gfCNCPoint3[4861] = {X 137.2439, Y 19.5606, Z -3.8333, A 0.000, B 0.000, C 0.000 }
gfCNCPoint3[4862] = {X 137.1370, Y 19.7298, Z -3.8333, A 0.000, B 0.000, C 0.000 }
gfCNCPoint3[4863] = {X 136.4975, Y 20.4532, Z -3.8333, A 0.000, B 0.000, C 0.000 }
gfCNCPoint3[4864] = {X 135.7033, Y 21.0023, Z -3.8333, A 0.000, B 0.000, C 0.000 }
gfCNCPoint3[4865] = {X 134.8007, Y 21.3450, Z -3.8333, A 0.000, B 0.000, C 0.000 }
gfCNCPoint3[4866] = {X 133.8422, Y 21.4615, Z -3.8333, A 0.000, B 0.000, C 0.000 }
gfCNCPoint3[4867] = {X 133.2006, Y 21.4615, Z -3.8333, A 0.000, B 0.000, C 0.000 }
gfCNCPoint3[4868] = {X 132.3106, Y 21.3612, Z -3.8333, A 0.000, B 0.000, C 0.000 }
gfCNCPoint3[4869] = {X 131.4651, Y 21.0654, Z -3.8333, A 0.000, B 0.000, C 0.000 }
gfCNCPoint3[4870] = {X 130.7067, Y 20.5889, Z -3.8333, A 0.000, B 0.000, C 0.000 }
gfCNCPoint3[4871] = {X 130.0733, Y 19.9555, Z -3.8333, A 0.000, B 0.000, C 0.000 }
gfCNCPoint3[4872] = {X 129.5968, Y 19.1971, Z -3.8333, A 0.000, B 0.000, C 0.000 }
gfCNCPoint3[4873] = {X 129.3009, Y 18.3516, Z -3.8333, A 0.000, B 0.000, C 0.000 }
gfCNCPoint3[4874] = {X 129.2006, Y 17.4615, Z -3.8333, A 0.000, B 0.000, C 0.000 }
gfCNCPoint3[4875] = {X 129.2006, Y 10.4835, Z -3.8333, A 0.000, B 0.000, C 0.000 }
gfCNCPoint3[4876] = {X 129.3009, Y 9.5934, Z -3.8333, A 0.000, B 0.000, C 0.000 }
gfCNCPoint3[4877] = {X 129.5968, Y 8.7480, Z -3.8333, A 0.000, B 0.000, C 0.000 }
gfCNCPoint3[4878] = {X 130.0733, Y 7.9895, Z -3.8333, A 0.000, B 0.000, C 0.000 }
gfCNCPoint3[4879] = {X 130.7067, Y 7.3562, Z -3.8333, A 0.000, B 0.000, C 0.000 }
gfCNCPoint3[4880] = {X 131.4651, Y 6.8796, Z -3.8333, A 0.000, B 0.000, C 0.000 }
gfCNCPoint3[4881] = {X 132.3106, Y 6.5838, Z -3.8333, A 0.000, B 0.000, C 0.000 }
gfCNCPoint3[4882] = {X 133.2007, Y 6.4835, Z -3.8333, A 0.000, B 0.000, C 0.000 }
gfCNCPoint3[4883] = {X 133.8833, Y 6.4837, Z -3.8333, A 0.000, B 0.000, C 0.000 }
gfCNCPoint3[4884] = {X 134.6794, Y 6.5721, Z -3.8333, A 0.000, B 0.000, C 0.000 }
gfCNCPoint3[4885] = {X 135.4419, Y 6.8173, Z -3.8333, A 0.000, B 0.000, C 0.000 }
gfCNCPoint3[4886] = {X 136.1403, Y 7.2095, Z -3.8333, A 0.000, B 0.000, C 0.000 }
gfCNCPoint3[4887] = {X 136.7465, Y 7.7329, Z -3.8333, A 0.000, B 0.000, C 0.000 }
gfCNCPoint3[4888] = {X 137.2363, Y 8.3667, Z -3.8333, A 0.000, B 0.000, C 0.000 }
gfCNCPoint3[4889] = {X 155.2276, Y 8.3667, Z -3.8333, A 0.000, B 0.000, C 0.000 }
gfCNCPoint3[4890] = {X 155.2814, Y 8.3748, Z -3.8333, A 0.000, B 0.000, C 0.000 }
gfCNCPoint3[4891] = {X 155.3392, Y 8.2843, Z -3.8333, A 0.000, B 0.000, C 0.000 }
gfCNCPoint3[4892] = {X 155.3994, Y 8.1955, Z -3.8333, A 0.000, B 0.000, C 0.000 }
gfCNCPoint3[4893] = {X 156.0387, Y 7.4799, Z -3.8333, A 0.000, B 0.000, C 0.000 }
gfCNCPoint3[4894] = {X 156.8301, Y 6.9372, Z -3.8333, A 0.000, B 0.000, C 0.000 }
gfCNCPoint3[4895] = {X 157.7279, Y 6.5986, Z -3.8333, A 0.000, B 0.000, C 0.000 }
gfCNCPoint3[4896] = {X 158.6806, Y 6.4835, Z -3.8333, A 0.000, B 0.000, C 0.000 }
gfCNCPoint3[4897] = {X 159.3739, Y 6.4839, Z -3.8333, A 0.000, B 0.000, C 0.000 }
gfCNCPoint3[4898] = {X 160.2554, Y 6.5939, Z -3.8333, A 0.000, B 0.000, C 0.000 }
gfCNCPoint3[4899] = {X 161.0909, Y 6.8959, Z -3.8333, A 0.000, B 0.000, C 0.000 }
gfCNCPoint3[4900] = {X 161.8391, Y 7.3747, Z -3.8333, A 0.000, B 0.000, C 0.000 }
gfCNCPoint3[4901] = {X 162.4632, Y 8.0070, Z -3.8333, A 0.000, B 0.000, C 0.000 }
gfCNCPoint3[4902] = {X 162.9324, Y 8.7613, Z -3.8333, A 0.000, B 0.000, C 0.000 }
gfCNCPoint3[4903] = {X 163.2234, Y 9.6007, Z -3.8333, A 0.000, B 0.000, C 0.000 }
gfCNCPoint3[4904] = {X 163.3221, Y 10.4835, Z -3.8333, A 0.000, B 0.000, C 0.000 }
gfCNCPoint3[4905] = {X 163.3221, Y 17.4615, Z -3.8333, A 0.000, B 0.000, C 0.000 }
gfCNCPoint3[4906] = {X 163.2218, Y 18.3516, Z -3.8333, A 0.000, B 0.000, C 0.000 }
gfCNCPoint3[4907] = {X 162.9260, Y 19.1971, Z -3.8333, A 0.000, B 0.000, C 0.000 }
gfCNCPoint3[4908] = {X 162.4494, Y 19.9555, Z -3.8333, A 0.000, B 0.000, C 0.000 }
gfCNCPoint3[4909] = {X 161.8160, Y 20.5889, Z -3.8333, A 0.000, B 0.000, C 0.000 }
gfCNCPoint3[4910] = {X 161.0576, Y 21.0654, Z -3.8333, A 0.000, B 0.000, C 0.000 }
gfCNCPoint3[4911] = {X 160.2121, Y 21.3613, Z -3.8333, A 0.000, B 0.000, C 0.000 }
gfCNCPoint3[4912] = {X 159.3221, Y 21.4615, Z -3.8333, A 0.000, B 0.000, C 0.000 }
gfCNCPoint3[4913] = {X 158.6805, Y 21.4615, Z -3.8333, A 0.000, B 0.000, C 0.000 }
gfCNCPoint3[4914] = {X 157.8711, Y 21.3759, Z -3.8333, A 0.000, B 0.000, C 0.000 }
gfCNCPoint3[4915] = {X 157.0952, Y 21.1295, Z -3.8333, A 0.000, B 0.000, C 0.000 }
gfCNCPoint3[4916] = {X 156.3846, Y 20.7325, Z -3.8333, A 0.000, B 0.000, C 0.000 }
gfCNCPoint3[4917] = {X 155.7681, Y 20.2010, Z -3.8333, A 0.000, B 0.000, C 0.000 }
gfCNCPoint3[4918] = {X 155.2709, Y 19.5565, Z -3.8333, A 0.000, B 0.000, C 0.000 }
gfCNCPoint3[4919] = {X 151.9562, Y 19.5580, Z -3.8333, A 0.000, B 0.000, C 0.000 }
gfCNCPoint3[4920] = {X 151.9548, Y 40.9999, Z -3.8333, A 0.000, B 0.000, C 0.000 }
gfCNCPoint3[4921] = {X 152.5009, Y 41.5878, Z -3.8333, A 0.000, B 0.000, C 0.000 }
gfCNCPoint3[4922] = {X 152.5884, Y 41.6922, Z -3.8333, A 0.000, B 0.000, C 0.000 }
gfCNCPoint3[4923] = {X 153.0743, Y 42.4563, Z -3.8333, A 0.000, B 0.000, C 0.000 }
gfCNCPoint3[4924] = {X 153.3776, Y 43.3095, Z -3.8333, A 0.000, B 0.000, C 0.000 }
gfCNCPoint3[4925] = {X 153.4831, Y 44.2089, Z -3.8333, A 0.000, B 0.000, C 0.000 }
gfCNCPoint3[4926] = {X 153.4829, Y 45.0384, Z -3.8333, A 0.000, B 0.000, C 0.000 }
gfCNCPoint3[4927] = {X 153.3753, Y 45.9222, Z -3.8333, A 0.000, B 0.000, C 0.000 }
gfCNCPoint3[4928] = {X 153.0750, Y 46.7602, Z -3.8333, A 0.000, B 0.000, C 0.000 }
gfCNCPoint3[4929] = {X 152.5967, Y 47.5111, Z -3.8333, A 0.000, B 0.000, C 0.000 }
gfCNCPoint3[4930] = {X 151.9642, Y 48.1376, Z -3.8333, A 0.000, B 0.000, C 0.000 }
gfCNCPoint3[4931] = {X 151.2087, Y 48.6086, Z -3.8333, A 0.000, B 0.000, C 0.000 }
gfCNCPoint3[4932] = {X 150.3678, Y 48.9009, Z -3.8333, A 0.000, B 0.000, C 0.000 }
gfCNCPoint3[4933] = {X 149.4831, Y 49.0000, Z -3.8333, A 0.000, B 0.000, C 0.000 }
gfCNCPoint3[4934] = {X 143.0396, Y 49.0000, Z -3.8333, A 0.000, B 0.000, C 0.000 }
gfCNCPoint3[4935] = {X 142.1495, Y 48.8997, Z -3.8333, A 0.000, B 0.000, C 0.000 }
gfCNCPoint3[4936] = {X 141.3041, Y 48.6039, Z -3.8333, A 0.000, B 0.000, C 0.000 }
gfCNCPoint3[4937] = {X 140.5457, Y 48.1273, Z -3.8333, A 0.000, B 0.000, C 0.000 }
gfCNCPoint3[4938] = {X 139.9123, Y 47.4939, Z -3.8333, A 0.000, B 0.000, C 0.000 }
gfCNCPoint3[4939] = {X 139.4357, Y 46.7355, Z -3.8333, A 0.000, B 0.000, C 0.000 }
gfCNCPoint3[4940] = {X 139.1399, Y 45.8900, Z -3.8333, A 0.000, B 0.000, C 0.000 }
gfCNCPoint3[4941] = {X 139.0396, Y 45.0000, Z -3.8333, A 0.000, B 0.000, C 0.000 }
gfCNCPoint3[4942] = {X 139.0400, Y 44.1538, Z -3.8333, A 0.000, B 0.000, C 0.000 }
gfCNCPoint3[4943] = {X 139.1506, Y 43.2730, Z -3.8333, A 0.000, B 0.000, C 0.000 }
gfCNCPoint3[4944] = {X 139.4528, Y 42.4382, Z -3.8333, A 0.000, B 0.000, C 0.000 }
gfCNCPoint3[4945] = {X 139.9317, Y 41.6907, Z -3.8333, A 0.000, B 0.000, C 0.000 }
gfCNCPoint3[4946] = {X 140.5636, Y 41.0672, Z -3.8333, A 0.000, B 0.000, C 0.000 }
gfCNCPoint3[4947] = {X 140.5636, Y 30.3965, Z -3.8333, A 0.000, B 0.000, C 0.000 }
gfCNCPoint3[4948] = {X 136.4836, Y 30.3965, Z -3.8333, A 0.000, B 0.000, C 0.000 }
gfCNCPoint3[4949] = {X 136.4836, Y 30.3965, Z -0.8333, A 0.000, B 0.000, C 0.000 }
gfCNCPoint3[4950] = {X 136.4836, Y 30.3965, Z 11.0000, A 0.000, B 0.000, C 0.000 }
gfCNCPoint3[4951] = {X 137.6636, Y 74.8930, Z 11.0000, A 0.000, B 0.000, C 0.000 }
gfCNCPoint3[4952] = {X 137.6636, Y 74.8930, Z -0.8333, A 0.000, B 0.000, C 0.000 }
gfCNCPoint3[4953] = {X 137.6636, Y 74.8930, Z -3.8333, A 0.000, B 0.000, C 0.000 }
gfCNCPoint3[4954] = {X 140.6803, Y 77.6400, Z -3.8333, A 0.000, B 0.000, C 0.000 }
gfCNCPoint3[4955] = {X 155.6326, Y 61.2204, Z -3.8333, A 0.000, B 0.000, C 0.000 }
gfCNCPoint3[4956] = {X 155.2775, Y 60.5146, Z -3.8333, A 0.000, B 0.000, C 0.000 }
gfCNCPoint3[4957] = {X 155.0569, Y 59.7559, Z -3.8333, A 0.000, B 0.000, C 0.000 }
gfCNCPoint3[4958] = {X 154.9781, Y 58.9697, Z -3.8333, A 0.000, B 0.000, C 0.000 }
gfCNCPoint3[4959] = {X 154.9780, Y 58.0000, Z -3.8333, A 0.000, B 0.000, C 0.000 }
gfCNCPoint3[4960] = {X 155.0863, Y 57.0387, Z -3.8333, A 0.000, B 0.000, C 0.000 }
gfCNCPoint3[4961] = {X 155.4058, Y 56.1256, Z -3.8333, A 0.000, B 0.000, C 0.000 }
gfCNCPoint3[4962] = {X 155.9204, Y 55.3065, Z -3.8333, A 0.000, B 0.000, C 0.000 }
gfCNCPoint3[4963] = {X 156.6045, Y 54.6225, Z -3.8333, A 0.000, B 0.000, C 0.000 }
gfCNCPoint3[4964] = {X 157.4236, Y 54.1078, Z -3.8333, A 0.000, B 0.000, C 0.000 }
gfCNCPoint3[4965] = {X 158.3367, Y 53.7883, Z -3.8333, A 0.000, B 0.000, C 0.000 }
gfCNCPoint3[4966] = {X 159.2980, Y 53.6800, Z -3.8333, A 0.000, B 0.000, C 0.000 }
gfCNCPoint3[4967] = {X 178.5335, Y 53.6800, Z -3.8333, A 0.000, B 0.000, C 0.000 }
gfCNCPoint3[4968] = {X 179.4948, Y 53.7883, Z -3.8333, A 0.000, B 0.000, C 0.000 }
gfCNCPoint3[4969] = {X 180.4079, Y 54.1078, Z -3.8333, A 0.000, B 0.000, C 0.000 }
gfCNCPoint3[4970] = {X 181.2270, Y 54.6225, Z -3.8333, A 0.000, B 0.000, C 0.000 }
gfCNCPoint3[4971] = {X 181.9110, Y 55.3065, Z -3.8333, A 0.000, B 0.000, C 0.000 }
gfCNCPoint3[4972] = {X 182.4257, Y 56.1256, Z -3.8333, A 0.000, B 0.000, C 0.000 }
gfCNCPoint3[4973] = {X 182.7452, Y 57.0387, Z -3.8333, A 0.000, B 0.000, C 0.000 }
gfCNCPoint3[4974] = {X 182.8535, Y 58.0000, Z -3.8333, A 0.000, B 0.000, C 0.000 }
gfCNCPoint3[4975] = {X 182.8535, Y 58.9342, Z -3.8333, A 0.000, B 0.000, C 0.000 }
gfCNCPoint3[4976] = {X 182.7808, Y 59.7234, Z -3.8333, A 0.000, B 0.000, C 0.000 }
gfCNCPoint3[4977] = {X 182.5651, Y 60.4860, Z -3.8333, A 0.000, B 0.000, C 0.000 }
gfCNCPoint3[4978] = {X 182.2138, Y 61.1963, Z -3.8333, A 0.000, B 0.000, C 0.000 }
gfCNCPoint3[4979] = {X 209.4784, Y 90.9541, Z -3.8333, A 0.000, B 0.000, C 0.000 }
gfCNCPoint3[4980] = {X 210.1358, Y 91.6211, Z -3.8333, A 0.000, B 0.000, C 0.000 }
gfCNCPoint3[4981] = {X 210.8401, Y 92.2385, Z -3.8333, A 0.000, B 0.000, C 0.000 }
gfCNCPoint3[4982] = {X 211.1140, Y 92.4118, Z -3.8333, A 0.000, B 0.000, C 0.000 }
gfCNCPoint3[4983] = {X 211.4211, Y 92.5156, Z -3.8333, A 0.000, B 0.000, C 0.000 }
gfCNCPoint3[4984] = {X 213.4039, Y 92.8249, Z -3.8333, A 0.000, B 0.000, C 0.000 }
gfCNCPoint3[4985] = {X 214.4546, Y 92.7361, Z -3.8333, A 0.000, B 0.000, C 0.000 }
gfCNCPoint3[4986] = {X 215.5072, Y 92.6759, Z -3.8333, A 0.000, B 0.000, C 0.000 }
gfCNCPoint3[4987] = {X 216.1773, Y 92.6027, Z -3.8333, A 0.000, B 0.000, C 0.000 }
gfCNCPoint3[4988] = {X 216.8225, Y 92.4076, Z -3.8333, A 0.000, B 0.000, C 0.000 }
gfCNCPoint3[4989] = {X 217.4210, Y 92.0974, Z -3.8333, A 0.000, B 0.000, C 0.000 }
gfCNCPoint3[4990] = {X 222.9613, Y 88.5219, Z -3.8333, A 0.000, B 0.000, C 0.000 }
gfCNCPoint3[4991] = {X 245.8284, Y 73.8995, Z -3.8333, A 0.000, B 0.000, C 0.000 }
gfCNCPoint3[4992] = {X 221.6305, Y 64.4034, Z -3.8333, A 0.000, B 0.000, C 0.000 }
gfCNCPoint3[4993] = {X 219.8632, Y 63.8117, Z -3.8333, A 0.000, B 0.000, C 0.000 }
gfCNCPoint3[4994] = {X 218.0397, Y 63.4261, Z -3.8333, A 0.000, B 0.000, C 0.000 }
gfCNCPoint3[4995] = {X 216.1842, Y 63.2516, Z -3.8333, A 0.000, B 0.000, C 0.000 }
gfCNCPoint3[4996] = {X 215.2523, Y 63.1173, Z -3.8333, A 0.000, B 0.000, C 0.000 }
gfCNCPoint3[4997] = {X 214.3717, Y 62.7843, Z -3.8333, A 0.000, B 0.000, C 0.000 }
gfCNCPoint3[4998] = {X 213.5841, Y 62.2684, Z -3.8333, A 0.000, B 0.000, C 0.000 }
gfCNCPoint3[4999] = {X 212.9270, Y 61.5942, Z -3.8333, A 0.000, B 0.000, C 0.000 }
gfCNCPoint3[5000] = {X 212.4315, Y 60.7936, Z -3.8333, A 0.000, B 0.000, C 0.000 }
gfCNCPoint3[5001] = {X 212.1213, Y 59.9047, Z -3.8333, A 0.000, B 0.000, C 0.000 }
gfCNCPoint3[5002] = {X 212.0110, Y 58.9697, Z -3.8333, A 0.000, B 0.000, C 0.000 }
gfCNCPoint3[5003] = {X 212.0108, Y 58.0000, Z -3.8333, A 0.000, B 0.000, C 0.000 }
gfCNCPoint3[5004] = {X 212.1191, Y 57.0387, Z -3.8333, A 0.000, B 0.000, C 0.000 }
gfCNCPoint3[5005] = {X 212.4386, Y 56.1256, Z -3.8333, A 0.000, B 0.000, C 0.000 }
gfCNCPoint3[5006] = {X 212.9533, Y 55.3065, Z -3.8333, A 0.000, B 0.000, C 0.000 }
gfCNCPoint3[5007] = {X 213.6373, Y 54.6225, Z -3.8333, A 0.000, B 0.000, C 0.000 }
gfCNCPoint3[5008] = {X 214.4564, Y 54.1078, Z -3.8333, A 0.000, B 0.000, C 0.000 }
gfCNCPoint3[5009] = {X 215.3695, Y 53.7883, Z -3.8333, A 0.000, B 0.000, C 0.000 }
gfCNCPoint3[5010] = {X 216.3308, Y 53.6800, Z -3.8333, A 0.000, B 0.000, C 0.000 }
gfCNCPoint3[5011] = {X 237.2617, Y 53.6800, Z -3.8333, A 0.000, B 0.000, C 0.000 }
gfCNCPoint3[5012] = {X 238.2230, Y 53.7883, Z -3.8333, A 0.000, B 0.000, C 0.000 }
gfCNCPoint3[5013] = {X 239.1361, Y 54.1078, Z -3.8333, A 0.000, B 0.000, C 0.000 }
gfCNCPoint3[5014] = {X 239.9552, Y 54.6225, Z -3.8333, A 0.000, B 0.000, C 0.000 }
gfCNCPoint3[5015] = {X 240.6392, Y 55.3065, Z -3.8333, A 0.000, B 0.000, C 0.000 }
gfCNCPoint3[5016] = {X 241.1539, Y 56.1256, Z -3.8333, A 0.000, B 0.000, C 0.000 }
gfCNCPoint3[5017] = {X 241.4734, Y 57.0387, Z -3.8333, A 0.000, B 0.000, C 0.000 }
gfCNCPoint3[5018] = {X 241.5817, Y 58.0000, Z -3.8333, A 0.000, B 0.000, C 0.000 }
gfCNCPoint3[5019] = {X 241.5817, Y 58.2325, Z -3.8333, A 0.000, B 0.000, C 0.000 }
gfCNCPoint3[5020] = {X 247.4883, Y 60.5350, Z -3.8333, A 0.000, B 0.000, C 0.000 }
gfCNCPoint3[5021] = {X 275.6332, Y 71.7024, Z -3.8333, A 0.000, B 0.000, C 0.000 }
gfCNCPoint3[5022] = {X 275.6341, Y 63.2124, Z -3.8333, A 0.000, B 0.000, C 0.000 }
gfCNCPoint3[5023] = {X 274.7824, Y 63.0033, Z -3.8333, A 0.000, B 0.000, C 0.000 }
gfCNCPoint3[5024] = {X 273.9904, Y 62.6266, Z -3.8333, A 0.000, B 0.000, C 0.000 }
gfCNCPoint3[5025] = {X 273.2909, Y 62.0976, Z -3.8333, A 0.000, B 0.000, C 0.000 }
gfCNCPoint3[5026] = {X 272.7126, Y 61.4383, Z -3.8333, A 0.000, B 0.000, C 0.000 }
gfCNCPoint3[5027] = {X 272.2794, Y 60.6758, Z -3.8333, A 0.000, B 0.000, C 0.000 }
gfCNCPoint3[5028] = {X 272.0091, Y 59.8415, Z -3.8333, A 0.000, B 0.000, C 0.000 }
gfCNCPoint3[5029] = {X 271.9128, Y 58.9697, Z -3.8333, A 0.000, B 0.000, C 0.000 }
gfCNCPoint3[5030] = {X 271.9127, Y 58.0000, Z -3.8333, A 0.000, B 0.000, C 0.000 }
gfCNCPoint3[5031] = {X 272.0210, Y 57.0387, Z -3.8333, A 0.000, B 0.000, C 0.000 }
gfCNCPoint3[5032] = {X 272.3405, Y 56.1256, Z -3.8333, A 0.000, B 0.000, C 0.000 }
gfCNCPoint3[5033] = {X 272.8552, Y 55.3065, Z -3.8333, A 0.000, B 0.000, C 0.000 }
gfCNCPoint3[5034] = {X 273.5392, Y 54.6225, Z -3.8333, A 0.000, B 0.000, C 0.000 }
gfCNCPoint3[5035] = {X 274.3583, Y 54.1078, Z -3.8333, A 0.000, B 0.000, C 0.000 }
gfCNCPoint3[5036] = {X 275.2714, Y 53.7883, Z -3.8333, A 0.000, B 0.000, C 0.000 }
gfCNCPoint3[5037] = {X 276.2327, Y 53.6800, Z -3.8333, A 0.000, B 0.000, C 0.000 }
gfCNCPoint3[5038] = {X 292.7731, Y 53.6800, Z -3.8333, A 0.000, B 0.000, C 0.000 }
gfCNCPoint3[5039] = {X 293.7344, Y 53.7883, Z -3.8333, A 0.000, B 0.000, C 0.000 }
gfCNCPoint3[5040] = {X 294.6475, Y 54.1078, Z -3.8333, A 0.000, B 0.000, C 0.000 }
gfCNCPoint3[5041] = {X 295.4666, Y 54.6225, Z -3.8333, A 0.000, B 0.000, C 0.000 }
gfCNCPoint3[5042] = {X 296.1506, Y 55.3065, Z -3.8333, A 0.000, B 0.000, C 0.000 }
gfCNCPoint3[5043] = {X 296.6653, Y 56.1256, Z -3.8333, A 0.000, B 0.000, C 0.000 }
gfCNCPoint3[5044] = {X 296.9848, Y 57.0387, Z -3.8333, A 0.000, B 0.000, C 0.000 }
gfCNCPoint3[5045] = {X 297.0931, Y 58.0000, Z -3.8333, A 0.000, B 0.000, C 0.000 }
gfCNCPoint3[5046] = {X 297.0931, Y 58.9351, Z -3.8333, A 0.000, B 0.000, C 0.000 }
gfCNCPoint3[5047] = {X 297.0007, Y 59.8116, Z -3.8333, A 0.000, B 0.000, C 0.000 }
gfCNCPoint3[5048] = {X 296.7330, Y 60.6513, Z -3.8333, A 0.000, B 0.000, C 0.000 }
gfCNCPoint3[5049] = {X 296.3011, Y 61.4195, Z -3.8333, A 0.000, B 0.000, C 0.000 }
gfCNCPoint3[5050] = {X 295.7228, Y 62.0846, Z -3.8333, A 0.000, B 0.000, C 0.000 }
gfCNCPoint3[5051] = {X 295.0220, Y 62.6189, Z -3.8333, A 0.000, B 0.000, C 0.000 }
gfCNCPoint3[5052] = {X 294.2276, Y 63.0006, Z -3.8333, A 0.000, B 0.000, C 0.000 }
gfCNCPoint3[5053] = {X 293.3725, Y 63.2138, Z -3.8333, A 0.000, B 0.000, C 0.000 }
gfCNCPoint3[5054] = {X 293.3844, Y 92.7814, Z -3.8333, A 0.000, B 0.000, C 0.000 }
gfCNCPoint3[5055] = {X 294.2369, Y 92.9989, Z -3.8333, A 0.000, B 0.000, C 0.000 }
gfCNCPoint3[5056] = {X 295.0282, Y 93.3833, Z -3.8333, A 0.000, B 0.000, C 0.000 }
gfCNCPoint3[5057] = {X 295.7261, Y 93.9190, Z -3.8333, A 0.000, B 0.000, C 0.000 }
gfCNCPoint3[5058] = {X 296.3020, Y 94.5841, Z -3.8333, A 0.000, B 0.000, C 0.000 }
gfCNCPoint3[5059] = {X 296.7324, Y 95.3514, Z -3.8333, A 0.000, B 0.000, C 0.000 }
gfCNCPoint3[5060] = {X 296.9998, Y 96.1896, Z -3.8333, A 0.000, B 0.000, C 0.000 }
gfCNCPoint3[5061] = {X 297.0931, Y 97.0645, Z -3.8333, A 0.000, B 0.000, C 0.000 }
gfCNCPoint3[5062] = {X 297.0931, Y 98.0000, Z -3.8333, A 0.000, B 0.000, C 0.000 }
gfCNCPoint3[5063] = {X 296.9848, Y 98.9613, Z -3.8333, A 0.000, B 0.000, C 0.000 }
gfCNCPoint3[5064] = {X 296.6653, Y 99.8744, Z -3.8333, A 0.000, B 0.000, C 0.000 }
gfCNCPoint3[5065] = {X 296.1506, Y 100.6935, Z -3.8333, A 0.000, B 0.000, C 0.000 }
gfCNCPoint3[5066] = {X 295.4666, Y 101.3775, Z -3.8333, A 0.000, B 0.000, C 0.000 }
gfCNCPoint3[5067] = {X 294.6475, Y 101.8922, Z -3.8333, A 0.000, B 0.000, C 0.000 }
gfCNCPoint3[5068] = {X 293.7344, Y 102.2117, Z -3.8333, A 0.000, B 0.000, C 0.000 }
gfCNCPoint3[5069] = {X 292.7731, Y 102.3200, Z -3.8333, A 0.000, B 0.000, C 0.000 }
gfCNCPoint3[5070] = {X 276.2327, Y 102.3200, Z -3.8333, A 0.000, B 0.000, C 0.000 }
gfCNCPoint3[5071] = {X 275.2714, Y 102.2117, Z -3.8333, A 0.000, B 0.000, C 0.000 }
gfCNCPoint3[5072] = {X 274.3583, Y 101.8922, Z -3.8333, A 0.000, B 0.000, C 0.000 }
gfCNCPoint3[5073] = {X 273.5392, Y 101.3775, Z -3.8333, A 0.000, B 0.000, C 0.000 }
gfCNCPoint3[5074] = {X 272.8552, Y 100.6935, Z -3.8333, A 0.000, B 0.000, C 0.000 }
gfCNCPoint3[5075] = {X 272.3405, Y 99.8744, Z -3.8333, A 0.000, B 0.000, C 0.000 }
gfCNCPoint3[5076] = {X 272.0210, Y 98.9613, Z -3.8333, A 0.000, B 0.000, C 0.000 }
gfCNCPoint3[5077] = {X 271.9127, Y 98.0000, Z -3.8333, A 0.000, B 0.000, C 0.000 }
gfCNCPoint3[5078] = {X 271.9127, Y 97.0659, Z -3.8333, A 0.000, B 0.000, C 0.000 }
gfCNCPoint3[5079] = {X 272.0026, Y 96.1891, Z -3.8333, A 0.000, B 0.000, C 0.000 }
gfCNCPoint3[5080] = {X 272.2686, Y 95.3488, Z -3.8333, A 0.000, B 0.000, C 0.000 }
gfCNCPoint3[5081] = {X 272.6996, Y 94.5800, Z -3.8333, A 0.000, B 0.000, C 0.000 }
gfCNCPoint3[5082] = {X 273.2777, Y 93.9146, Z -3.8333, A 0.000, B 0.000, C 0.000 }
gfCNCPoint3[5083] = {X 273.9788, Y 93.3805, Z -3.8333, A 0.000, B 0.000, C 0.000 }
gfCNCPoint3[5084] = {X 274.7737, Y 92.9997, Z -3.8333, A 0.000, B 0.000, C 0.000 }
gfCNCPoint3[5085] = {X 275.6294, Y 92.7883, Z -3.8333, A 0.000, B 0.000, C 0.000 }
gfCNCPoint3[5086] = {X 275.6294, Y 85.5950, Z -3.8333, A 0.000, B 0.000, C 0.000 }
gfCNCPoint3[5087] = {X 262.6396, Y 80.5030, Z -3.8333, A 0.000, B 0.000, C 0.000 }
gfCNCPoint3[5088] = {X 262.2767, Y 80.7316, Z -3.8333, A 0.000, B 0.000, C 0.000 }
gfCNCPoint3[5089] = {X 237.7964, Y 96.5881, Z -3.8333, A 0.000, B 0.000, C 0.000 }
gfCNCPoint3[5090] = {X 237.7998, Y 97.0648, Z -3.8333, A 0.000, B 0.000, C 0.000 }
gfCNCPoint3[5091] = {X 237.7998, Y 98.0000, Z -3.8333, A 0.000, B 0.000, C 0.000 }
gfCNCPoint3[5092] = {X 237.6915, Y 98.9613, Z -3.8333, A 0.000, B 0.000, C 0.000 }
gfCNCPoint3[5093] = {X 237.3720, Y 99.8744, Z -3.8333, A 0.000, B 0.000, C 0.000 }
gfCNCPoint3[5094] = {X 236.8573, Y 100.6935, Z -3.8333, A 0.000, B 0.000, C 0.000 }
gfCNCPoint3[5095] = {X 236.1733, Y 101.3775, Z -3.8333, A 0.000, B 0.000, C 0.000 }
gfCNCPoint3[5096] = {X 235.3542, Y 101.8922, Z -3.8333, A 0.000, B 0.000, C 0.000 }
gfCNCPoint3[5097] = {X 234.4411, Y 102.2117, Z -3.8333, A 0.000, B 0.000, C 0.000 }
gfCNCPoint3[5098] = {X 233.4798, Y 102.3200, Z -3.8333, A 0.000, B 0.000, C 0.000 }
gfCNCPoint3[5099] = {X 214.1790, Y 102.3200, Z -3.8333, A 0.000, B 0.000, C 0.000 }
gfCNCPoint3[5100] = {X 213.7862, Y 102.3021, Z -3.8333, A 0.000, B 0.000, C 0.000 }
gfCNCPoint3[5101] = {X 213.3966, Y 102.2485, Z -3.8333, A 0.000, B 0.000, C 0.000 }
gfCNCPoint3[5102] = {X 213.0070, Y 102.3021, Z -3.8333, A 0.000, B 0.000, C 0.000 }
gfCNCPoint3[5103] = {X 212.6141, Y 102.3200, Z -3.8333, A 0.000, B 0.000, C 0.000 }
gfCNCPoint3[5104] = {X 194.9870, Y 102.3200, Z -3.8333, A 0.000, B 0.000, C 0.000 }
gfCNCPoint3[5105] = {X 194.0257, Y 102.2117, Z -3.8333, A 0.000, B 0.000, C 0.000 }
gfCNCPoint3[5106] = {X 193.1126, Y 101.8922, Z -3.8333, A 0.000, B 0.000, C 0.000 }
gfCNCPoint3[5107] = {X 192.2935, Y 101.3775, Z -3.8333, A 0.000, B 0.000, C 0.000 }
gfCNCPoint3[5108] = {X 191.6094, Y 100.6935, Z -3.8333, A 0.000, B 0.000, C 0.000 }
gfCNCPoint3[5109] = {X 191.0948, Y 99.8744, Z -3.8333, A 0.000, B 0.000, C 0.000 }
gfCNCPoint3[5110] = {X 190.7753, Y 98.9613, Z -3.8333, A 0.000, B 0.000, C 0.000 }
gfCNCPoint3[5111] = {X 190.6670, Y 98.0000, Z -3.8333, A 0.000, B 0.000, C 0.000 }
gfCNCPoint3[5112] = {X 190.6670, Y 97.0659, Z -3.8333, A 0.000, B 0.000, C 0.000 }
gfCNCPoint3[5113] = {X 190.7727, Y 96.1162, Z -3.8333, A 0.000, B 0.000, C 0.000 }
gfCNCPoint3[5114] = {X 191.0846, Y 95.2129, Z -3.8333, A 0.000, B 0.000, C 0.000 }
gfCNCPoint3[5115] = {X 191.5874, Y 94.4003, Z -3.8333, A 0.000, B 0.000, C 0.000 }
gfCNCPoint3[5116] = {X 188.5647, Y 91.1002, Z -3.8333, A 0.000, B 0.000, C 0.000 }
gfCNCPoint3[5117] = {X 150.0898, Y 91.1002, Z -3.8333, A 0.000, B 0.000, C 0.000 }
gfCNCPoint3[5118] = {X 147.1448, Y 94.3629, Z -3.8333, A 0.000, B 0.000, C 0.000 }
gfCNCPoint3[5119] = {X 147.6636, Y 95.1842, Z -3.8333, A 0.000, B 0.000, C 0.000 }
gfCNCPoint3[5120] = {X 147.9870, Y 96.1001, Z -3.8333, A 0.000, B 0.000, C 0.000 }
gfCNCPoint3[5121] = {X 148.0991, Y 97.0649, Z -3.8333, A 0.000, B 0.000, C 0.000 }
gfCNCPoint3[5122] = {X 148.0991, Y 98.0000, Z -3.8333, A 0.000, B 0.000, C 0.000 }
gfCNCPoint3[5123] = {X 147.9908, Y 98.9613, Z -3.8333, A 0.000, B 0.000, C 0.000 }
gfCNCPoint3[5124] = {X 147.6713, Y 99.8744, Z -3.8333, A 0.000, B 0.000, C 0.000 }
gfCNCPoint3[5125] = {X 147.1566, Y 100.6935, Z -3.8333, A 0.000, B 0.000, C 0.000 }
gfCNCPoint3[5126] = {X 146.4726, Y 101.3775, Z -3.8333, A 0.000, B 0.000, C 0.000 }
gfCNCPoint3[5127] = {X 145.6535, Y 101.8922, Z -3.8333, A 0.000, B 0.000, C 0.000 }
gfCNCPoint3[5128] = {X 144.7404, Y 102.2117, Z -3.8333, A 0.000, B 0.000, C 0.000 }
gfCNCPoint3[5129] = {X 143.7791, Y 102.3200, Z -3.8333, A 0.000, B 0.000, C 0.000 }
gfCNCPoint3[5130] = {X 125.0000, Y 102.3200, Z -3.8333, A 0.000, B 0.000, C 0.000 }
gfCNCPoint3[5131] = {X 124.0387, Y 102.2117, Z -3.8333, A 0.000, B 0.000, C 0.000 }
gfCNCPoint3[5132] = {X 123.1256, Y 101.8922, Z -3.8333, A 0.000, B 0.000, C 0.000 }
gfCNCPoint3[5133] = {X 122.3065, Y 101.3775, Z -3.8333, A 0.000, B 0.000, C 0.000 }
gfCNCPoint3[5134] = {X 121.6225, Y 100.6935, Z -3.8333, A 0.000, B 0.000, C 0.000 }
gfCNCPoint3[5135] = {X 121.1078, Y 99.8744, Z -3.8333, A 0.000, B 0.000, C 0.000 }
gfCNCPoint3[5136] = {X 120.7883, Y 98.9613, Z -3.8333, A 0.000, B 0.000, C 0.000 }
gfCNCPoint3[5137] = {X 120.6800, Y 98.0000, Z -3.8333, A 0.000, B 0.000, C 0.000 }
gfCNCPoint3[5138] = {X 120.6800, Y 97.0659, Z -3.8333, A 0.000, B 0.000, C 0.000 }
gfCNCPoint3[5139] = {X 120.7832, Y 96.1272, Z -3.8333, A 0.000, B 0.000, C 0.000 }
gfCNCPoint3[5140] = {X 121.0880, Y 95.2334, Z -3.8333, A 0.000, B 0.000, C 0.000 }
gfCNCPoint3[5141] = {X 121.5797, Y 94.4271, Z -3.8333, A 0.000, B 0.000, C 0.000 }
gfCNCPoint3[5142] = {X 122.2348, Y 93.7469, Z -3.8333, A 0.000, B 0.000, C 0.000 }
gfCNCPoint3[5143] = {X 123.0221, Y 93.2253, Z -3.8333, A 0.000, B 0.000, C 0.000 }
gfCNCPoint3[5144] = {X 123.9039, Y 92.8873, Z -3.8333, A 0.000, B 0.000, C 0.000 }
gfCNCPoint3[5145] = {X 124.8381, Y 92.7490, Z -3.8333, A 0.000, B 0.000, C 0.000 }
gfCNCPoint3[5146] = {X 124.8820, Y 92.7321, Z -3.8333, A 0.000, B 0.000, C 0.000 }
gfCNCPoint3[5147] = {X 124.9279, Y 92.7218, Z -3.8333, A 0.000, B 0.000, C 0.000 }
gfCNCPoint3[5148] = {X 125.4494, Y 92.6444, Z -3.8333, A 0.000, B 0.000, C 0.000 }
gfCNCPoint3[5149] = {X 126.2806, Y 92.5046, Z -3.8333, A 0.000, B 0.000, C 0.000 }
gfCNCPoint3[5150] = {X 127.1003, Y 92.3081, Z -3.8333, A 0.000, B 0.000, C 0.000 }
gfCNCPoint3[5151] = {X 128.3219, Y 91.1565, Z -3.8333, A 0.000, B 0.000, C 0.000 }
gfCNCPoint3[5152] = {X 129.4793, Y 89.9402, Z -3.8333, A 0.000, B 0.000, C 0.000 }
gfCNCPoint3[5153] = {X 140.6803, Y 77.6400, Z -3.8333, A 0.000, B 0.000, C 0.000 }
gfCNCPoint3[5154] = {X 137.7228, Y 74.9468, Z -3.8333, A 0.000, B 0.000, C 0.000 }
gfCNCPoint3[5155] = {X 140.7394, Y 77.6939, Z -3.8333, A 0.000, B 0.000, C 0.000 }
gfCNCPoint3[5156] = {X 155.7328, Y 61.2291, Z -3.8333, A 0.000, B 0.000, C 0.000 }
gfCNCPoint3[5157] = {X 155.3668, Y 60.5227, Z -3.8333, A 0.000, B 0.000, C 0.000 }
gfCNCPoint3[5158] = {X 155.1393, Y 59.7605, Z -3.8333, A 0.000, B 0.000, C 0.000 }
gfCNCPoint3[5159] = {X 155.0581, Y 58.9691, Z -3.8333, A 0.000, B 0.000, C 0.000 }
gfCNCPoint3[5160] = {X 155.0580, Y 58.0000, Z -3.8333, A 0.000, B 0.000, C 0.000 }
gfCNCPoint3[5161] = {X 155.1643, Y 57.0565, Z -3.8333, A 0.000, B 0.000, C 0.000 }
gfCNCPoint3[5162] = {X 155.4778, Y 56.1603, Z -3.8333, A 0.000, B 0.000, C 0.000 }
gfCNCPoint3[5163] = {X 155.9830, Y 55.3564, Z -3.8333, A 0.000, B 0.000, C 0.000 }
gfCNCPoint3[5164] = {X 156.6544, Y 54.6850, Z -3.8333, A 0.000, B 0.000, C 0.000 }
gfCNCPoint3[5165] = {X 157.4583, Y 54.1799, Z -3.8333, A 0.000, B 0.000, C 0.000 }
gfCNCPoint3[5166] = {X 158.3545, Y 53.8663, Z -3.8333, A 0.000, B 0.000, C 0.000 }
gfCNCPoint3[5167] = {X 159.2980, Y 53.7600, Z -3.8333, A 0.000, B 0.000, C 0.000 }
gfCNCPoint3[5168] = {X 178.5335, Y 53.7600, Z -3.8333, A 0.000, B 0.000, C 0.000 }
gfCNCPoint3[5169] = {X 179.4770, Y 53.8663, Z -3.8333, A 0.000, B 0.000, C 0.000 }
gfCNCPoint3[5170] = {X 180.3732, Y 54.1799, Z -3.8333, A 0.000, B 0.000, C 0.000 }
gfCNCPoint3[5171] = {X 181.1771, Y 54.6850, Z -3.8333, A 0.000, B 0.000, C 0.000 }
gfCNCPoint3[5172] = {X 181.8485, Y 55.3564, Z -3.8333, A 0.000, B 0.000, C 0.000 }
gfCNCPoint3[5173] = {X 182.3536, Y 56.1603, Z -3.8333, A 0.000, B 0.000, C 0.000 }
gfCNCPoint3[5174] = {X 182.6672, Y 57.0565, Z -3.8333, A 0.000, B 0.000, C 0.000 }
gfCNCPoint3[5175] = {X 182.7735, Y 58.0000, Z -3.8333, A 0.000, B 0.000, C 0.000 }
gfCNCPoint3[5176] = {X 182.7735, Y 58.9342, Z -3.8333, A 0.000, B 0.000, C 0.000 }
gfCNCPoint3[5177] = {X 182.6984, Y 59.7285, Z -3.8333, A 0.000, B 0.000, C 0.000 }
gfCNCPoint3[5178] = {X 182.4759, Y 60.4946, Z -3.8333, A 0.000, B 0.000, C 0.000 }
gfCNCPoint3[5179] = {X 182.1137, Y 61.2055, Z -3.8333, A 0.000, B 0.000, C 0.000 }
gfCNCPoint3[5180] = {X 209.4194, Y 91.0081, Z -3.8333, A 0.000, B 0.000, C 0.000 }
gfCNCPoint3[5181] = {X 210.0809, Y 91.6793, Z -3.8333, A 0.000, B 0.000, C 0.000 }
gfCNCPoint3[5182] = {X 210.7896, Y 92.3006, Z -3.8333, A 0.000, B 0.000, C 0.000 }
gfCNCPoint3[5183] = {X 211.0805, Y 92.4845, Z -3.8333, A 0.000, B 0.000, C 0.000 }
gfCNCPoint3[5184] = {X 211.4067, Y 92.5943, Z -3.8333, A 0.000, B 0.000, C 0.000 }
gfCNCPoint3[5185] = {X 213.4016, Y 92.9055, Z -3.8333, A 0.000, B 0.000, C 0.000 }
gfCNCPoint3[5186] = {X 214.4546, Y 92.8163, Z -3.8333, A 0.000, B 0.000, C 0.000 }
gfCNCPoint3[5187] = {X 215.5096, Y 92.7559, Z -3.8333, A 0.000, B 0.000, C 0.000 }
gfCNCPoint3[5188] = {X 216.1940, Y 92.6809, Z -3.8333, A 0.000, B 0.000, C 0.000 }
gfCNCPoint3[5189] = {X 216.8531, Y 92.4816, Z -3.8333, A 0.000, B 0.000, C 0.000 }
gfCNCPoint3[5190] = {X 217.4643, Y 92.1647, Z -3.8333, A 0.000, B 0.000, C 0.000 }
gfCNCPoint3[5191] = {X 223.0046, Y 88.5892, Z -3.8333, A 0.000, B 0.000, C 0.000 }
gfCNCPoint3[5192] = {X 246.0037, Y 73.8824, Z -3.8333, A 0.000, B 0.000, C 0.000 }
gfCNCPoint3[5193] = {X 221.6602, Y 64.3291, Z -3.8333, A 0.000, B 0.000, C 0.000 }
gfCNCPoint3[5194] = {X 219.8842, Y 63.7345, Z -3.8333, A 0.000, B 0.000, C 0.000 }
gfCNCPoint3[5195] = {X 218.0518, Y 63.3470, Z -3.8333, A 0.000, B 0.000, C 0.000 }
gfCNCPoint3[5196] = {X 216.1871, Y 63.1716, Z -3.8333, A 0.000, B 0.000, C 0.000 }
gfCNCPoint3[5197] = {X 215.2725, Y 63.0399, Z -3.8333, A 0.000, B 0.000, C 0.000 }
gfCNCPoint3[5198] = {X 214.4081, Y 62.7131, Z -3.8333, A 0.000, B 0.000, C 0.000 }
gfCNCPoint3[5199] = {X 213.6351, Y 62.2068, Z -3.8333, A 0.000, B 0.000, C 0.000 }
gfCNCPoint3[5200] = {X 212.9901, Y 61.5450, Z -3.8333, A 0.000, B 0.000, C 0.000 }
gfCNCPoint3[5201] = {X 212.5038, Y 60.7593, Z -3.8333, A 0.000, B 0.000, C 0.000 }
gfCNCPoint3[5202] = {X 212.1992, Y 59.8868, Z -3.8333, A 0.000, B 0.000, C 0.000 }
gfCNCPoint3[5203] = {X 212.0910, Y 58.9691, Z -3.8333, A 0.000, B 0.000, C 0.000 }
gfCNCPoint3[5204] = {X 212.0908, Y 58.0000, Z -3.8333, A 0.000, B 0.000, C 0.000 }
gfCNCPoint3[5205] = {X 212.1971, Y 57.0565, Z -3.8333, A 0.000, B 0.000, C 0.000 }
gfCNCPoint3[5206] = {X 212.5107, Y 56.1603, Z -3.8333, A 0.000, B 0.000, C 0.000 }
gfCNCPoint3[5207] = {X 213.0158, Y 55.3564, Z -3.8333, A 0.000, B 0.000, C 0.000 }
gfCNCPoint3[5208] = {X 213.6872, Y 54.6850, Z -3.8333, A 0.000, B 0.000, C 0.000 }
gfCNCPoint3[5209] = {X 214.4911, Y 54.1799, Z -3.8333, A 0.000, B 0.000, C 0.000 }
gfCNCPoint3[5210] = {X 215.3873, Y 53.8663, Z -3.8333, A 0.000, B 0.000, C 0.000 }
gfCNCPoint3[5211] = {X 216.3308, Y 53.7600, Z -3.8333, A 0.000, B 0.000, C 0.000 }
gfCNCPoint3[5212] = {X 237.2617, Y 53.7600, Z -3.8333, A 0.000, B 0.000, C 0.000 }
gfCNCPoint3[5213] = {X 238.2052, Y 53.8663, Z -3.8333, A 0.000, B 0.000, C 0.000 }
gfCNCPoint3[5214] = {X 239.1014, Y 54.1799, Z -3.8333, A 0.000, B 0.000, C 0.000 }
gfCNCPoint3[5215] = {X 239.9053, Y 54.6850, Z -3.8333, A 0.000, B 0.000, C 0.000 }
gfCNCPoint3[5216] = {X 240.5767, Y 55.3564, Z -3.8333, A 0.000, B 0.000, C 0.000 }
gfCNCPoint3[5217] = {X 241.0818, Y 56.1603, Z -3.8333, A 0.000, B 0.000, C 0.000 }
gfCNCPoint3[5218] = {X 241.3954, Y 57.0565, Z -3.8333, A 0.000, B 0.000, C 0.000 }
gfCNCPoint3[5219] = {X 241.5017, Y 58.0000, Z -3.8333, A 0.000, B 0.000, C 0.000 }
gfCNCPoint3[5220] = {X 241.5017, Y 58.2871, Z -3.8333, A 0.000, B 0.000, C 0.000 }
gfCNCPoint3[5221] = {X 247.4591, Y 60.6094, Z -3.8333, A 0.000, B 0.000, C 0.000 }
gfCNCPoint3[5222] = {X 275.7132, Y 71.8203, Z -3.8333, A 0.000, B 0.000, C 0.000 }
gfCNCPoint3[5223] = {X 275.7141, Y 63.1422, Z -3.8333, A 0.000, B 0.000, C 0.000 }
gfCNCPoint3[5224] = {X 274.8655, Y 62.9476, Z -3.8333, A 0.000, B 0.000, C 0.000 }
gfCNCPoint3[5225] = {X 274.0745, Y 62.5837, Z -3.8333, A 0.000, B 0.000, C 0.000 }
gfCNCPoint3[5226] = {X 273.3746, Y 62.0660, Z -3.8333, A 0.000, B 0.000, C 0.000 }
gfCNCPoint3[5227] = {X 272.7951, Y 61.4162, Z -3.8333, A 0.000, B 0.000, C 0.000 }
gfCNCPoint3[5228] = {X 272.3606, Y 60.6617, Z -3.8333, A 0.000, B 0.000, C 0.000 }
gfCNCPoint3[5229] = {X 272.0894, Y 59.8344, Z -3.8333, A 0.000, B 0.000, C 0.000 }
gfCNCPoint3[5230] = {X 271.9928, Y 58.9691, Z -3.8333, A 0.000, B 0.000, C 0.000 }
gfCNCPoint3[5231] = {X 271.9927, Y 58.0000, Z -3.8333, A 0.000, B 0.000, C 0.000 }
gfCNCPoint3[5232] = {X 272.0990, Y 57.0565, Z -3.8333, A 0.000, B 0.000, C 0.000 }
gfCNCPoint3[5233] = {X 272.4126, Y 56.1603, Z -3.8333, A 0.000, B 0.000, C 0.000 }
gfCNCPoint3[5234] = {X 272.9177, Y 55.3564, Z -3.8333, A 0.000, B 0.000, C 0.000 }
gfCNCPoint3[5235] = {X 273.5891, Y 54.6850, Z -3.8333, A 0.000, B 0.000, C 0.000 }
gfCNCPoint3[5236] = {X 274.3930, Y 54.1799, Z -3.8333, A 0.000, B 0.000, C 0.000 }
gfCNCPoint3[5237] = {X 275.2892, Y 53.8663, Z -3.8333, A 0.000, B 0.000, C 0.000 }
gfCNCPoint3[5238] = {X 276.2327, Y 53.7600, Z -3.8333, A 0.000, B 0.000, C 0.000 }
gfCNCPoint3[5239] = {X 292.7731, Y 53.7600, Z -3.8333, A 0.000, B 0.000, C 0.000 }
gfCNCPoint3[5240] = {X 293.7166, Y 53.8663, Z -3.8333, A 0.000, B 0.000, C 0.000 }
gfCNCPoint3[5241] = {X 294.6128, Y 54.1799, Z -3.8333, A 0.000, B 0.000, C 0.000 }
gfCNCPoint3[5242] = {X 295.4167, Y 54.6850, Z -3.8333, A 0.000, B 0.000, C 0.000 }
gfCNCPoint3[5243] = {X 296.0881, Y 55.3564, Z -3.8333, A 0.000, B 0.000, C 0.000 }
gfCNCPoint3[5244] = {X 296.5932, Y 56.1603, Z -3.8333, A 0.000, B 0.000, C 0.000 }
gfCNCPoint3[5245] = {X 296.9068, Y 57.0565, Z -3.8333, A 0.000, B 0.000, C 0.000 }
gfCNCPoint3[5246] = {X 297.0131, Y 58.0000, Z -3.8333, A 0.000, B 0.000, C 0.000 }
gfCNCPoint3[5247] = {X 297.0131, Y 58.9349, Z -3.8333, A 0.000, B 0.000, C 0.000 }
gfCNCPoint3[5248] = {X 296.9204, Y 59.8045, Z -3.8333, A 0.000, B 0.000, C 0.000 }
gfCNCPoint3[5249] = {X 296.6520, Y 60.6369, Z -3.8333, A 0.000, B 0.000, C 0.000 }
gfCNCPoint3[5250] = {X 296.2191, Y 61.3969, Z -3.8333, A 0.000, B 0.000, C 0.000 }
gfCNCPoint3[5251] = {X 295.6400, Y 62.0523, Z -3.8333, A 0.000, B 0.000, C 0.000 }
gfCNCPoint3[5252] = {X 294.9392, Y 62.5755, Z -3.8333, A 0.000, B 0.000, C 0.000 }
gfCNCPoint3[5253] = {X 294.1463, Y 62.9445, Z -3.8333, A 0.000, B 0.000, C 0.000 }
gfCNCPoint3[5254] = {X 293.2946, Y 63.1436, Z -3.8333, A 0.000, B 0.000, C 0.000 }
gfCNCPoint3[5255] = {X 293.3044, Y 92.8509, Z -3.8333, A 0.000, B 0.000, C 0.000 }
gfCNCPoint3[5256] = {X 294.1538, Y 93.0541, Z -3.8333, A 0.000, B 0.000, C 0.000 }
gfCNCPoint3[5257] = {X 294.9442, Y 93.4258, Z -3.8333, A 0.000, B 0.000, C 0.000 }
gfCNCPoint3[5258] = {X 295.6425, Y 93.9504, Z -3.8333, A 0.000, B 0.000, C 0.000 }
gfCNCPoint3[5259] = {X 296.2195, Y 94.6060, Z -3.8333, A 0.000, B 0.000, C 0.000 }
gfCNCPoint3[5260] = {X 296.6512, Y 95.3653, Z -3.8333, A 0.000, B 0.000, C 0.000 }
gfCNCPoint3[5261] = {X 296.9194, Y 96.1965, Z -3.8333, A 0.000, B 0.000, C 0.000 }
gfCNCPoint3[5262] = {X 297.0131, Y 97.0649, Z -3.8333, A 0.000, B 0.000, C 0.000 }
gfCNCPoint3[5263] = {X 297.0131, Y 98.0000, Z -3.8333, A 0.000, B 0.000, C 0.000 }
gfCNCPoint3[5264] = {X 296.9068, Y 98.9435, Z -3.8333, A 0.000, B 0.000, C 0.000 }
gfCNCPoint3[5265] = {X 296.5932, Y 99.8397, Z -3.8333, A 0.000, B 0.000, C 0.000 }
gfCNCPoint3[5266] = {X 296.0881, Y 100.6436, Z -3.8333, A 0.000, B 0.000, C 0.000 }
gfCNCPoint3[5267] = {X 295.4167, Y 101.3150, Z -3.8333, A 0.000, B 0.000, C 0.000 }
gfCNCPoint3[5268] = {X 294.6128, Y 101.8201, Z -3.8333, A 0.000, B 0.000, C 0.000 }
gfCNCPoint3[5269] = {X 293.7166, Y 102.1337, Z -3.8333, A 0.000, B 0.000, C 0.000 }
gfCNCPoint3[5270] = {X 292.7731, Y 102.2400, Z -3.8333, A 0.000, B 0.000, C 0.000 }
gfCNCPoint3[5271] = {X 276.2327, Y 102.2400, Z -3.8333, A 0.000, B 0.000, C 0.000 }
gfCNCPoint3[5272] = {X 275.2892, Y 102.1337, Z -3.8333, A 0.000, B 0.000, C 0.000 }
gfCNCPoint3[5273] = {X 274.3930, Y 101.8201, Z -3.8333, A 0.000, B 0.000, C 0.000 }
gfCNCPoint3[5274] = {X 273.5891, Y 101.3150, Z -3.8333, A 0.000, B 0.000, C 0.000 }
gfCNCPoint3[5275] = {X 272.9177, Y 100.6436, Z -3.8333, A 0.000, B 0.000, C 0.000 }
gfCNCPoint3[5276] = {X 272.4126, Y 99.8397, Z -3.8333, A 0.000, B 0.000, C 0.000 }
gfCNCPoint3[5277] = {X 272.0990, Y 98.9435, Z -3.8333, A 0.000, B 0.000, C 0.000 }
gfCNCPoint3[5278] = {X 271.9927, Y 98.0000, Z -3.8333, A 0.000, B 0.000, C 0.000 }
gfCNCPoint3[5279] = {X 271.9927, Y 97.0659, Z -3.8333, A 0.000, B 0.000, C 0.000 }
gfCNCPoint3[5280] = {X 272.0830, Y 96.1956, Z -3.8333, A 0.000, B 0.000, C 0.000 }
gfCNCPoint3[5281] = {X 272.3500, Y 95.3624, Z -3.8333, A 0.000, B 0.000, C 0.000 }
gfCNCPoint3[5282] = {X 272.7823, Y 94.6017, Z -3.8333, A 0.000, B 0.000, C 0.000 }
gfCNCPoint3[5283] = {X 273.3615, Y 93.9460, Z -3.8333, A 0.000, B 0.000, C 0.000 }
gfCNCPoint3[5284] = {X 274.0630, Y 93.4231, Z -3.8333, A 0.000, B 0.000, C 0.000 }
gfCNCPoint3[5285] = {X 274.8569, Y 93.0553, Z -3.8333, A 0.000, B 0.000, C 0.000 }
gfCNCPoint3[5286] = {X 275.7094, Y 92.8584, Z -3.8333, A 0.000, B 0.000, C 0.000 }
gfCNCPoint3[5287] = {X 275.7094, Y 85.5404, Z -3.8333, A 0.000, B 0.000, C 0.000 }
gfCNCPoint3[5288] = {X 262.6312, Y 80.4137, Z -3.8333, A 0.000, B 0.000, C 0.000 }
gfCNCPoint3[5289] = {X 262.2336, Y 80.6642, Z -3.8333, A 0.000, B 0.000, C 0.000 }
gfCNCPoint3[5290] = {X 237.7161, Y 96.5448, Z -3.8333, A 0.000, B 0.000, C 0.000 }
gfCNCPoint3[5291] = {X 237.7198, Y 97.0651, Z -3.8333, A 0.000, B 0.000, C 0.000 }
gfCNCPoint3[5292] = {X 237.7198, Y 98.0000, Z -3.8333, A 0.000, B 0.000, C 0.000 }
gfCNCPoint3[5293] = {X 237.6135, Y 98.9435, Z -3.8333, A 0.000, B 0.000, C 0.000 }
gfCNCPoint3[5294] = {X 237.2999, Y 99.8397, Z -3.8333, A 0.000, B 0.000, C 0.000 }
gfCNCPoint3[5295] = {X 236.7948, Y 100.6436, Z -3.8333, A 0.000, B 0.000, C 0.000 }
gfCNCPoint3[5296] = {X 236.1234, Y 101.3150, Z -3.8333, A 0.000, B 0.000, C 0.000 }
gfCNCPoint3[5297] = {X 235.3195, Y 101.8201, Z -3.8333, A 0.000, B 0.000, C 0.000 }
gfCNCPoint3[5298] = {X 234.4233, Y 102.1337, Z -3.8333, A 0.000, B 0.000, C 0.000 }
gfCNCPoint3[5299] = {X 233.4798, Y 102.2400, Z -3.8333, A 0.000, B 0.000, C 0.000 }
gfCNCPoint3[5300] = {X 214.1790, Y 102.2400, Z -3.8333, A 0.000, B 0.000, C 0.000 }
gfCNCPoint3[5301] = {X 213.7861, Y 102.2218, Z -3.8333, A 0.000, B 0.000, C 0.000 }
gfCNCPoint3[5302] = {X 213.3966, Y 102.1672, Z -3.8333, A 0.000, B 0.000, C 0.000 }
gfCNCPoint3[5303] = {X 213.0070, Y 102.2218, Z -3.8333, A 0.000, B 0.000, C 0.000 }
gfCNCPoint3[5304] = {X 212.6141, Y 102.2400, Z -3.8333, A 0.000, B 0.000, C 0.000 }
gfCNCPoint3[5305] = {X 194.9870, Y 102.2400, Z -3.8333, A 0.000, B 0.000, C 0.000 }
gfCNCPoint3[5306] = {X 194.0435, Y 102.1337, Z -3.8333, A 0.000, B 0.000, C 0.000 }
gfCNCPoint3[5307] = {X 193.1473, Y 101.8201, Z -3.8333, A 0.000, B 0.000, C 0.000 }
gfCNCPoint3[5308] = {X 192.3434, Y 101.3150, Z -3.8333, A 0.000, B 0.000, C 0.000 }
gfCNCPoint3[5309] = {X 191.6720, Y 100.6436, Z -3.8333, A 0.000, B 0.000, C 0.000 }
gfCNCPoint3[5310] = {X 191.1669, Y 99.8397, Z -3.8333, A 0.000, B 0.000, C 0.000 }
gfCNCPoint3[5311] = {X 190.8533, Y 98.9435, Z -3.8333, A 0.000, B 0.000, C 0.000 }
gfCNCPoint3[5312] = {X 190.7470, Y 98.0000, Z -3.8333, A 0.000, B 0.000, C 0.000 }
gfCNCPoint3[5313] = {X 190.7470, Y 97.0659, Z -3.8333, A 0.000, B 0.000, C 0.000 }
gfCNCPoint3[5314] = {X 190.8557, Y 96.1118, Z -3.8333, A 0.000, B 0.000, C 0.000 }
gfCNCPoint3[5315] = {X 191.1764, Y 95.2065, Z -3.8333, A 0.000, B 0.000, C 0.000 }
gfCNCPoint3[5316] = {X 191.6926, Y 94.3967, Z -3.8333, A 0.000, B 0.000, C 0.000 }
gfCNCPoint3[5317] = {X 188.5999, Y 91.0202, Z -3.8333, A 0.000, B 0.000, C 0.000 }
gfCNCPoint3[5318] = {X 150.0543, Y 91.0202, Z -3.8333, A 0.000, B 0.000, C 0.000 }
gfCNCPoint3[5319] = {X 147.0395, Y 94.3603, Z -3.8333, A 0.000, B 0.000, C 0.000 }
gfCNCPoint3[5320] = {X 147.5716, Y 95.1784, Z -3.8333, A 0.000, B 0.000, C 0.000 }
gfCNCPoint3[5321] = {X 147.9039, Y 96.0961, Z -3.8333, A 0.000, B 0.000, C 0.000 }
gfCNCPoint3[5322] = {X 148.0191, Y 97.0652, Z -3.8333, A 0.000, B 0.000, C 0.000 }
gfCNCPoint3[5323] = {X 148.0191, Y 98.0000, Z -3.8333, A 0.000, B 0.000, C 0.000 }
gfCNCPoint3[5324] = {X 147.9128, Y 98.9435, Z -3.8333, A 0.000, B 0.000, C 0.000 }
gfCNCPoint3[5325] = {X 147.5992, Y 99.8397, Z -3.8333, A 0.000, B 0.000, C 0.000 }
gfCNCPoint3[5326] = {X 147.0941, Y 100.6436, Z -3.8333, A 0.000, B 0.000, C 0.000 }
gfCNCPoint3[5327] = {X 146.4227, Y 101.3150, Z -3.8333, A 0.000, B 0.000, C 0.000 }
gfCNCPoint3[5328] = {X 145.6188, Y 101.8201, Z -3.8333, A 0.000, B 0.000, C 0.000 }
gfCNCPoint3[5329] = {X 144.7226, Y 102.1337, Z -3.8333, A 0.000, B 0.000, C 0.000 }
gfCNCPoint3[5330] = {X 143.7791, Y 102.2400, Z -3.8333, A 0.000, B 0.000, C 0.000 }
gfCNCPoint3[5331] = {X 125.0000, Y 102.2400, Z -3.8333, A 0.000, B 0.000, C 0.000 }
gfCNCPoint3[5332] = {X 124.0565, Y 102.1337, Z -3.8333, A 0.000, B 0.000, C 0.000 }
gfCNCPoint3[5333] = {X 123.1603, Y 101.8201, Z -3.8333, A 0.000, B 0.000, C 0.000 }
gfCNCPoint3[5334] = {X 122.3564, Y 101.3150, Z -3.8333, A 0.000, B 0.000, C 0.000 }
gfCNCPoint3[5335] = {X 121.6850, Y 100.6436, Z -3.8333, A 0.000, B 0.000, C 0.000 }
gfCNCPoint3[5336] = {X 121.1799, Y 99.8397, Z -3.8333, A 0.000, B 0.000, C 0.000 }
gfCNCPoint3[5337] = {X 120.8663, Y 98.9435, Z -3.8333, A 0.000, B 0.000, C 0.000 }
gfCNCPoint3[5338] = {X 120.7600, Y 98.0000, Z -3.8333, A 0.000, B 0.000, C 0.000 }
gfCNCPoint3[5339] = {X 120.7600, Y 97.0659, Z -3.8333, A 0.000, B 0.000, C 0.000 }
gfCNCPoint3[5340] = {X 120.8619, Y 96.1422, Z -3.8333, A 0.000, B 0.000, C 0.000 }
gfCNCPoint3[5341] = {X 121.1625, Y 95.2628, Z -3.8333, A 0.000, B 0.000, C 0.000 }
gfCNCPoint3[5342] = {X 121.6476, Y 94.4700, Z -3.8333, A 0.000, B 0.000, C 0.000 }
gfCNCPoint3[5343] = {X 122.2937, Y 93.8020, Z -3.8333, A 0.000, B 0.000, C 0.000 }
gfCNCPoint3[5344] = {X 123.0699, Y 93.2907, Z -3.8333, A 0.000, B 0.000, C 0.000 }
gfCNCPoint3[5345] = {X 123.9387, Y 92.9609, Z -3.8333, A 0.000, B 0.000, C 0.000 }
gfCNCPoint3[5346] = {X 124.8586, Y 92.8283, Z -3.8333, A 0.000, B 0.000, C 0.000 }
gfCNCPoint3[5347] = {X 124.8979, Y 92.8110, Z -3.8333, A 0.000, B 0.000, C 0.000 }
gfCNCPoint3[5348] = {X 124.9396, Y 92.8009, Z -3.8333, A 0.000, B 0.000, C 0.000 }
gfCNCPoint3[5349] = {X 125.4606, Y 92.7236, Z -3.8333, A 0.000, B 0.000, C 0.000 }
gfCNCPoint3[5350] = {X 126.3061, Y 92.5810, Z -3.8333, A 0.000, B 0.000, C 0.000 }
gfCNCPoint3[5351] = {X 127.1396, Y 92.3802, Z -3.8333, A 0.000, B 0.000, C 0.000 }
gfCNCPoint3[5352] = {X 128.3718, Y 91.2198, Z -3.8333, A 0.000, B 0.000, C 0.000 }
gfCNCPoint3[5353] = {X 129.5387, Y 89.9938, Z -3.8333, A 0.000, B 0.000, C 0.000 }
gfCNCPoint3[5354] = {X 140.7394, Y 77.6939, Z -3.8333, A 0.000, B 0.000, C 0.000 }
gfCNCPoint3[5355] = {X 137.7819, Y 75.0007, Z -3.8333, A 0.000, B 0.000, C 0.000 }
gfCNCPoint3[5356] = {X 140.7986, Y 77.7477, Z -3.8333, A 0.000, B 0.000, C 0.000 }
gfCNCPoint3[5357] = {X 155.8337, Y 61.2372, Z -3.8333, A 0.000, B 0.000, C 0.000 }
gfCNCPoint3[5358] = {X 155.4565, Y 60.5306, Z -3.8333, A 0.000, B 0.000, C 0.000 }
gfCNCPoint3[5359] = {X 155.2218, Y 59.7649, Z -3.8333, A 0.000, B 0.000, C 0.000 }
gfCNCPoint3[5360] = {X 155.1381, Y 58.9684, Z -3.8333, A 0.000, B 0.000, C 0.000 }
gfCNCPoint3[5361] = {X 155.1380, Y 58.0000, Z -3.8333, A 0.000, B 0.000, C 0.000 }
gfCNCPoint3[5362] = {X 155.2423, Y 57.0743, Z -3.8333, A 0.000, B 0.000, C 0.000 }
gfCNCPoint3[5363] = {X 155.5499, Y 56.1950, Z -3.8333, A 0.000, B 0.000, C 0.000 }
gfCNCPoint3[5364] = {X 156.0455, Y 55.4063, Z -3.8333, A 0.000, B 0.000, C 0.000 }
gfCNCPoint3[5365] = {X 156.7042, Y 54.7476, Z -3.8333, A 0.000, B 0.000, C 0.000 }
gfCNCPoint3[5366] = {X 157.4930, Y 54.2520, Z -3.8333, A 0.000, B 0.000, C 0.000 }
gfCNCPoint3[5367] = {X 158.3723, Y 53.9443, Z -3.8333, A 0.000, B 0.000, C 0.000 }
gfCNCPoint3[5368] = {X 159.2980, Y 53.8400, Z -3.8333, A 0.000, B 0.000, C 0.000 }
gfCNCPoint3[5369] = {X 178.5335, Y 53.8400, Z -3.8333, A 0.000, B 0.000, C 0.000 }
gfCNCPoint3[5370] = {X 179.4592, Y 53.9443, Z -3.8333, A 0.000, B 0.000, C 0.000 }
gfCNCPoint3[5371] = {X 180.3385, Y 54.2520, Z -3.8333, A 0.000, B 0.000, C 0.000 }
gfCNCPoint3[5372] = {X 181.1272, Y 54.7476, Z -3.8333, A 0.000, B 0.000, C 0.000 }
gfCNCPoint3[5373] = {X 181.7859, Y 55.4063, Z -3.8333, A 0.000, B 0.000, C 0.000 }
gfCNCPoint3[5374] = {X 182.2815, Y 56.1950, Z -3.8333, A 0.000, B 0.000, C 0.000 }
gfCNCPoint3[5375] = {X 182.5892, Y 57.0743, Z -3.8333, A 0.000, B 0.000, C 0.000 }
gfCNCPoint3[5376] = {X 182.6935, Y 58.0000, Z -3.8333, A 0.000, B 0.000, C 0.000 }
gfCNCPoint3[5377] = {X 182.6935, Y 58.9342, Z -3.8333, A 0.000, B 0.000, C 0.000 }
gfCNCPoint3[5378] = {X 182.6160, Y 59.7335, Z -3.8333, A 0.000, B 0.000, C 0.000 }
gfCNCPoint3[5379] = {X 182.3863, Y 60.5030, Z -3.8333, A 0.000, B 0.000, C 0.000 }
gfCNCPoint3[5380] = {X 182.0130, Y 61.2141, Z -3.8333, A 0.000, B 0.000, C 0.000 }
gfCNCPoint3[5381] = {X 209.3604, Y 91.0621, Z -3.8333, A 0.000, B 0.000, C 0.000 }
gfCNCPoint3[5382] = {X 210.0260, Y 91.7375, Z -3.8333, A 0.000, B 0.000, C 0.000 }
gfCNCPoint3[5383] = {X 210.7391, Y 92.3626, Z -3.8333, A 0.000, B 0.000, C 0.000 }
gfCNCPoint3[5384] = {X 211.0470, Y 92.5572, Z -3.8333, A 0.000, B 0.000, C 0.000 }
gfCNCPoint3[5385] = {X 211.3924, Y 92.6730, Z -3.8333, A 0.000, B 0.000, C 0.000 }
gfCNCPoint3[5386] = {X 213.3994, Y 92.9861, Z -3.8333, A 0.000, B 0.000, C 0.000 }
gfCNCPoint3[5387] = {X 214.4547, Y 92.8965, Z -3.8333, A 0.000, B 0.000, C 0.000 }
gfCNCPoint3[5388] = {X 215.5121, Y 92.8358, Z -3.8333, A 0.000, B 0.000, C 0.000 }
gfCNCPoint3[5389] = {X 216.2108, Y 92.7591, Z -3.8333, A 0.000, B 0.000, C 0.000 }
gfCNCPoint3[5390] = {X 216.8836, Y 92.5555, Z -3.8333, A 0.000, B 0.000, C 0.000 }
gfCNCPoint3[5391] = {X 217.5077, Y 92.2319, Z -3.8333, A 0.000, B 0.000, C 0.000 }
gfCNCPoint3[5392] = {X 223.0478, Y 88.6566, Z -3.8333, A 0.000, B 0.000, C 0.000 }
gfCNCPoint3[5393] = {X 246.1791, Y 73.8652, Z -3.8333, A 0.000, B 0.000, C 0.000 }
gfCNCPoint3[5394] = {X 221.6899, Y 64.2548, Z -3.8333, A 0.000, B 0.000, C 0.000 }
gfCNCPoint3[5395] = {X 219.9052, Y 63.6573, Z -3.8333, A 0.000, B 0.000, C 0.000 }
gfCNCPoint3[5396] = {X 218.0638, Y 63.2679, Z -3.8333, A 0.000, B 0.000, C 0.000 }
gfCNCPoint3[5397] = {X 216.1900, Y 63.0917, Z -3.8333, A 0.000, B 0.000, C 0.000 }
gfCNCPoint3[5398] = {X 215.2926, Y 62.9624, Z -3.8333, A 0.000, B 0.000, C 0.000 }
gfCNCPoint3[5399] = {X 214.4445, Y 62.6418, Z -3.8333, A 0.000, B 0.000, C 0.000 }
gfCNCPoint3[5400] = {X 213.6860, Y 62.1451, Z -3.8333, A 0.000, B 0.000, C 0.000 }
gfCNCPoint3[5401] = {X 213.0532, Y 61.4958, Z -3.8333, A 0.000, B 0.000, C 0.000 }
gfCNCPoint3[5402] = {X 212.5760, Y 60.7249, Z -3.8333, A 0.000, B 0.000, C 0.000 }
gfCNCPoint3[5403] = {X 212.2772, Y 59.8688, Z -3.8333, A 0.000, B 0.000, C 0.000 }
gfCNCPoint3[5404] = {X 212.1710, Y 58.9684, Z -3.8333, A 0.000, B 0.000, C 0.000 }
gfCNCPoint3[5405] = {X 212.1708, Y 58.0000, Z -3.8333, A 0.000, B 0.000, C 0.000 }
gfCNCPoint3[5406] = {X 212.2751, Y 57.0743, Z -3.8333, A 0.000, B 0.000, C 0.000 }
gfCNCPoint3[5407] = {X 212.5828, Y 56.1950, Z -3.8333, A 0.000, B 0.000, C 0.000 }
gfCNCPoint3[5408] = {X 213.0784, Y 55.4063, Z -3.8333, A 0.000, B 0.000, C 0.000 }
gfCNCPoint3[5409] = {X 213.7371, Y 54.7476, Z -3.8333, A 0.000, B 0.000, C 0.000 }
gfCNCPoint3[5410] = {X 214.5259, Y 54.2520, Z -3.8333, A 0.000, B 0.000, C 0.000 }
gfCNCPoint3[5411] = {X 215.4051, Y 53.9443, Z -3.8333, A 0.000, B 0.000, C 0.000 }
gfCNCPoint3[5412] = {X 216.3308, Y 53.8400, Z -3.8333, A 0.000, B 0.000, C 0.000 }
gfCNCPoint3[5413] = {X 237.2617, Y 53.8400, Z -3.8333, A 0.000, B 0.000, C 0.000 }
gfCNCPoint3[5414] = {X 238.1874, Y 53.9443, Z -3.8333, A 0.000, B 0.000, C 0.000 }
gfCNCPoint3[5415] = {X 239.0666, Y 54.2520, Z -3.8333, A 0.000, B 0.000, C 0.000 }
gfCNCPoint3[5416] = {X 239.8554, Y 54.7476, Z -3.8333, A 0.000, B 0.000, C 0.000 }
gfCNCPoint3[5417] = {X 240.5141, Y 55.4063, Z -3.8333, A 0.000, B 0.000, C 0.000 }
gfCNCPoint3[5418] = {X 241.0097, Y 56.1950, Z -3.8333, A 0.000, B 0.000, C 0.000 }
gfCNCPoint3[5419] = {X 241.3174, Y 57.0743, Z -3.8333, A 0.000, B 0.000, C 0.000 }
gfCNCPoint3[5420] = {X 241.4217, Y 58.0000, Z -3.8333, A 0.000, B 0.000, C 0.000 }
gfCNCPoint3[5421] = {X 241.4217, Y 58.3418, Z -3.8333, A 0.000, B 0.000, C 0.000 }
gfCNCPoint3[5422] = {X 247.4298, Y 60.6839, Z -3.8333, A 0.000, B 0.000, C 0.000 }
gfCNCPoint3[5423] = {X 275.7932, Y 71.9381, Z -3.8333, A 0.000, B 0.000, C 0.000 }
gfCNCPoint3[5424] = {X 275.7941, Y 63.0709, Z -3.8333, A 0.000, B 0.000, C 0.000 }
gfCNCPoint3[5425] = {X 275.6917, Y 63.0587, Z -3.8333, A 0.000, B 0.000, C 0.000 }
gfCNCPoint3[5426] = {X 275.5896, Y 63.0441, Z -3.8333, A 0.000, B 0.000, C 0.000 }
gfCNCPoint3[5427] = {X 274.6520, Y 62.7821, Z -3.8333, A 0.000, B 0.000, C 0.000 }
gfCNCPoint3[5428] = {X 273.8010, Y 62.3093, Z -3.8333, A 0.000, B 0.000, C 0.000 }
gfCNCPoint3[5429] = {X 273.0831, Y 61.6518, Z -3.8333, A 0.000, B 0.000, C 0.000 }
gfCNCPoint3[5430] = {X 272.5378, Y 60.8454, Z -3.8333, A 0.000, B 0.000, C 0.000 }
gfCNCPoint3[5431] = {X 272.1947, Y 59.9343, Z -3.8333, A 0.000, B 0.000, C 0.000 }
gfCNCPoint3[5432] = {X 272.0728, Y 58.9684, Z -3.8333, A 0.000, B 0.000, C 0.000 }
gfCNCPoint3[5433] = {X 272.0727, Y 58.0000, Z -3.8333, A 0.000, B 0.000, C 0.000 }
gfCNCPoint3[5434] = {X 272.1770, Y 57.0743, Z -3.8333, A 0.000, B 0.000, C 0.000 }
gfCNCPoint3[5435] = {X 272.4847, Y 56.1950, Z -3.8333, A 0.000, B 0.000, C 0.000 }
gfCNCPoint3[5436] = {X 272.9803, Y 55.4063, Z -3.8333, A 0.000, B 0.000, C 0.000 }
gfCNCPoint3[5437] = {X 273.6390, Y 54.7476, Z -3.8333, A 0.000, B 0.000, C 0.000 }
gfCNCPoint3[5438] = {X 274.4277, Y 54.2520, Z -3.8333, A 0.000, B 0.000, C 0.000 }
gfCNCPoint3[5439] = {X 275.3070, Y 53.9443, Z -3.8333, A 0.000, B 0.000, C 0.000 }
gfCNCPoint3[5440] = {X 276.2327, Y 53.8400, Z -3.8333, A 0.000, B 0.000, C 0.000 }
gfCNCPoint3[5441] = {X 292.7731, Y 53.8400, Z -3.8333, A 0.000, B 0.000, C 0.000 }
gfCNCPoint3[5442] = {X 293.6988, Y 53.9443, Z -3.8333, A 0.000, B 0.000, C 0.000 }
gfCNCPoint3[5443] = {X 294.5780, Y 54.2520, Z -3.8333, A 0.000, B 0.000, C 0.000 }
gfCNCPoint3[5444] = {X 295.3668, Y 54.7476, Z -3.8333, A 0.000, B 0.000, C 0.000 }
gfCNCPoint3[5445] = {X 296.0255, Y 55.4063, Z -3.8333, A 0.000, B 0.000, C 0.000 }
gfCNCPoint3[5446] = {X 296.5211, Y 56.1950, Z -3.8333, A 0.000, B 0.000, C 0.000 }
gfCNCPoint3[5447] = {X 296.8288, Y 57.0743, Z -3.8333, A 0.000, B 0.000, C 0.000 }
gfCNCPoint3[5448] = {X 296.9331, Y 58.0000, Z -3.8333, A 0.000, B 0.000, C 0.000 }
gfCNCPoint3[5449] = {X 296.9331, Y 58.9346, Z -3.8333, A 0.000, B 0.000, C 0.000 }
gfCNCPoint3[5450] = {X 296.8153, Y 59.9063, Z -3.8333, A 0.000, B 0.000, C 0.000 }
gfCNCPoint3[5451] = {X 296.4745, Y 60.8239, Z -3.8333, A 0.000, B 0.000, C 0.000 }
gfCNCPoint3[5452] = {X 295.9296, Y 61.6369, Z -3.8333, A 0.000, B 0.000, C 0.000 }
gfCNCPoint3[5453] = {X 295.2104, Y 62.3008, Z -3.8333, A 0.000, B 0.000, C 0.000 }
gfCNCPoint3[5454] = {X 294.3564, Y 62.7792, Z -3.8333, A 0.000, B 0.000, C 0.000 }
gfCNCPoint3[5455] = {X 293.4146, Y 63.0456, Z -3.8333, A 0.000, B 0.000, C 0.000 }
gfCNCPoint3[5456] = {X 293.3182, Y 63.0598, Z -3.8333, A 0.000, B 0.000, C 0.000 }
gfCNCPoint3[5457] = {X 293.2214, Y 63.0718, Z -3.8333, A 0.000, B 0.000, C 0.000 }
gfCNCPoint3[5458] = {X 293.2124, Y 63.1620, Z -3.8333, A 0.000, B 0.000, C 0.000 }
gfCNCPoint3[5459] = {X 293.2244, Y 92.9216, Z -3.8333, A 0.000, B 0.000, C 0.000 }
gfCNCPoint3[5460] = {X 293.3193, Y 92.9337, Z -3.8333, A 0.000, B 0.000, C 0.000 }
gfCNCPoint3[5461] = {X 293.4139, Y 92.9480, Z -3.8333, A 0.000, B 0.000, C 0.000 }
gfCNCPoint3[5462] = {X 294.3554, Y 93.2171, Z -3.8333, A 0.000, B 0.000, C 0.000 }
gfCNCPoint3[5463] = {X 295.2088, Y 93.6972, Z -3.8333, A 0.000, B 0.000, C 0.000 }
gfCNCPoint3[5464] = {X 295.9275, Y 94.3621, Z -3.8333, A 0.000, B 0.000, C 0.000 }
gfCNCPoint3[5465] = {X 296.4725, Y 95.1756, Z -3.8333, A 0.000, B 0.000, C 0.000 }
gfCNCPoint3[5466] = {X 296.8139, Y 96.0934, Z -3.8333, A 0.000, B 0.000, C 0.000 }
gfCNCPoint3[5467] = {X 296.9331, Y 97.0653, Z -3.8333, A 0.000, B 0.000, C 0.000 }
gfCNCPoint3[5468] = {X 296.9331, Y 98.0000, Z -3.8333, A 0.000, B 0.000, C 0.000 }
gfCNCPoint3[5469] = {X 296.8288, Y 98.9257, Z -3.8333, A 0.000, B 0.000, C 0.000 }
gfCNCPoint3[5470] = {X 296.5211, Y 99.8050, Z -3.8333, A 0.000, B 0.000, C 0.000 }
gfCNCPoint3[5471] = {X 296.0255, Y 100.5937, Z -3.8333, A 0.000, B 0.000, C 0.000 }
gfCNCPoint3[5472] = {X 295.3668, Y 101.2524, Z -3.8333, A 0.000, B 0.000, C 0.000 }
gfCNCPoint3[5473] = {X 294.5780, Y 101.7480, Z -3.8333, A 0.000, B 0.000, C 0.000 }
gfCNCPoint3[5474] = {X 293.6988, Y 102.0557, Z -3.8333, A 0.000, B 0.000, C 0.000 }
gfCNCPoint3[5475] = {X 292.7731, Y 102.1600, Z -3.8333, A 0.000, B 0.000, C 0.000 }
gfCNCPoint3[5476] = {X 276.2327, Y 102.1600, Z -3.8333, A 0.000, B 0.000, C 0.000 }
gfCNCPoint3[5477] = {X 275.3070, Y 102.0557, Z -3.8333, A 0.000, B 0.000, C 0.000 }
gfCNCPoint3[5478] = {X 274.4277, Y 101.7480, Z -3.8333, A 0.000, B 0.000, C 0.000 }
gfCNCPoint3[5479] = {X 273.6390, Y 101.2524, Z -3.8333, A 0.000, B 0.000, C 0.000 }
gfCNCPoint3[5480] = {X 272.9803, Y 100.5937, Z -3.8333, A 0.000, B 0.000, C 0.000 }
gfCNCPoint3[5481] = {X 272.4847, Y 99.8050, Z -3.8333, A 0.000, B 0.000, C 0.000 }
gfCNCPoint3[5482] = {X 272.1770, Y 98.9257, Z -3.8333, A 0.000, B 0.000, C 0.000 }
gfCNCPoint3[5483] = {X 272.0727, Y 98.0000, Z -3.8333, A 0.000, B 0.000, C 0.000 }
gfCNCPoint3[5484] = {X 272.0727, Y 97.0659, Z -3.8333, A 0.000, B 0.000, C 0.000 }
gfCNCPoint3[5485] = {X 272.1633, Y 96.2022, Z -3.8333, A 0.000, B 0.000, C 0.000 }
gfCNCPoint3[5486] = {X 272.4314, Y 95.3761, Z -3.8333, A 0.000, B 0.000, C 0.000 }
gfCNCPoint3[5487] = {X 272.8650, Y 94.6237, Z -3.8333, A 0.000, B 0.000, C 0.000 }
gfCNCPoint3[5488] = {X 273.4455, Y 93.9777, Z -3.8333, A 0.000, B 0.000, C 0.000 }
gfCNCPoint3[5489] = {X 274.1474, Y 93.4663, Z -3.8333, A 0.000, B 0.000, C 0.000 }
gfCNCPoint3[5490] = {X 274.9402, Y 93.1118, Z -3.8333, A 0.000, B 0.000, C 0.000 }
gfCNCPoint3[5491] = {X 275.7894, Y 92.9296, Z -3.8333, A 0.000, B 0.000, C 0.000 }
gfCNCPoint3[5492] = {X 275.7894, Y 85.4858, Z -3.8333, A 0.000, B 0.000, C 0.000 }
gfCNCPoint3[5493] = {X 262.6227, Y 80.3245, Z -3.8333, A 0.000, B 0.000, C 0.000 }
gfCNCPoint3[5494] = {X 262.1905, Y 80.5968, Z -3.8333, A 0.000, B 0.000, C 0.000 }
gfCNCPoint3[5495] = {X 237.6358, Y 96.5015, Z -3.8333, A 0.000, B 0.000, C 0.000 }
gfCNCPoint3[5496] = {X 237.6398, Y 97.0653, Z -3.8333, A 0.000, B 0.000, C 0.000 }
gfCNCPoint3[5497] = {X 237.6398, Y 98.0000, Z -3.8333, A 0.000, B 0.000, C 0.000 }
gfCNCPoint3[5498] = {X 237.5355, Y 98.9257, Z -3.8333, A 0.000, B 0.000, C 0.000 }
gfCNCPoint3[5499] = {X 237.2278, Y 99.8050, Z -3.8333, A 0.000, B 0.000, C 0.000 }
gfCNCPoint3[5500] = {X 236.7322, Y 100.5937, Z -3.8333, A 0.000, B 0.000, C 0.000 }
gfCNCPoint3[5501] = {X 236.0735, Y 101.2524, Z -3.8333, A 0.000, B 0.000, C 0.000 }
gfCNCPoint3[5502] = {X 235.2847, Y 101.7480, Z -3.8333, A 0.000, B 0.000, C 0.000 }
gfCNCPoint3[5503] = {X 234.4055, Y 102.0557, Z -3.8333, A 0.000, B 0.000, C 0.000 }
gfCNCPoint3[5504] = {X 233.4798, Y 102.1600, Z -3.8333, A 0.000, B 0.000, C 0.000 }
gfCNCPoint3[5505] = {X 214.1790, Y 102.1600, Z -3.8333, A 0.000, B 0.000, C 0.000 }
gfCNCPoint3[5506] = {X 213.7860, Y 102.1414, Z -3.8333, A 0.000, B 0.000, C 0.000 }
gfCNCPoint3[5507] = {X 213.3966, Y 102.0857, Z -3.8333, A 0.000, B 0.000, C 0.000 }
gfCNCPoint3[5508] = {X 213.0071, Y 102.1414, Z -3.8333, A 0.000, B 0.000, C 0.000 }
gfCNCPoint3[5509] = {X 212.6141, Y 102.1600, Z -3.8333, A 0.000, B 0.000, C 0.000 }
gfCNCPoint3[5510] = {X 194.9870, Y 102.1600, Z -3.8333, A 0.000, B 0.000, C 0.000 }
gfCNCPoint3[5511] = {X 194.0613, Y 102.0557, Z -3.8333, A 0.000, B 0.000, C 0.000 }
gfCNCPoint3[5512] = {X 193.1820, Y 101.7480, Z -3.8333, A 0.000, B 0.000, C 0.000 }
gfCNCPoint3[5513] = {X 192.3932, Y 101.2524, Z -3.8333, A 0.000, B 0.000, C 0.000 }
gfCNCPoint3[5514] = {X 191.7345, Y 100.5937, Z -3.8333, A 0.000, B 0.000, C 0.000 }
gfCNCPoint3[5515] = {X 191.2389, Y 99.8050, Z -3.8333, A 0.000, B 0.000, C 0.000 }
gfCNCPoint3[5516] = {X 190.9313, Y 98.9257, Z -3.8333, A 0.000, B 0.000, C 0.000 }
gfCNCPoint3[5517] = {X 190.8270, Y 98.0000, Z -3.8333, A 0.000, B 0.000, C 0.000 }
gfCNCPoint3[5518] = {X 190.8270, Y 97.0659, Z -3.8333, A 0.000, B 0.000, C 0.000 }
gfCNCPoint3[5519] = {X 190.9241, Y 96.1723, Z -3.8333, A 0.000, B 0.000, C 0.000 }
gfCNCPoint3[5520] = {X 191.2109, Y 95.3203, Z -3.8333, A 0.000, B 0.000, C 0.000 }
gfCNCPoint3[5521] = {X 191.6741, Y 94.5499, Z -3.8333, A 0.000, B 0.000, C 0.000 }
gfCNCPoint3[5522] = {X 191.7354, Y 94.4712, Z -3.8333, A 0.000, B 0.000, C 0.000 }
gfCNCPoint3[5523] = {X 191.7986, Y 94.3939, Z -3.8333, A 0.000, B 0.000, C 0.000 }
gfCNCPoint3[5524] = {X 188.6351, Y 90.9402, Z -3.8333, A 0.000, B 0.000, C 0.000 }
gfCNCPoint3[5525] = {X 150.0187, Y 90.9402, Z -3.8333, A 0.000, B 0.000, C 0.000 }
gfCNCPoint3[5526] = {X 146.9334, Y 94.3584, Z -3.8333, A 0.000, B 0.000, C 0.000 }
gfCNCPoint3[5527] = {X 147.4792, Y 95.1730, Z -3.8333, A 0.000, B 0.000, C 0.000 }
gfCNCPoint3[5528] = {X 147.8207, Y 96.0921, Z -3.8333, A 0.000, B 0.000, C 0.000 }
gfCNCPoint3[5529] = {X 147.9391, Y 97.0655, Z -3.8333, A 0.000, B 0.000, C 0.000 }
gfCNCPoint3[5530] = {X 147.9391, Y 98.0000, Z -3.8333, A 0.000, B 0.000, C 0.000 }
gfCNCPoint3[5531] = {X 147.8348, Y 98.9257, Z -3.8333, A 0.000, B 0.000, C 0.000 }
gfCNCPoint3[5532] = {X 147.5271, Y 99.8050, Z -3.8333, A 0.000, B 0.000, C 0.000 }
gfCNCPoint3[5533] = {X 147.0315, Y 100.5937, Z -3.8333, A 0.000, B 0.000, C 0.000 }
gfCNCPoint3[5534] = {X 146.3728, Y 101.2524, Z -3.8333, A 0.000, B 0.000, C 0.000 }
gfCNCPoint3[5535] = {X 145.5841, Y 101.7480, Z -3.8333, A 0.000, B 0.000, C 0.000 }
gfCNCPoint3[5536] = {X 144.7048, Y 102.0557, Z -3.8333, A 0.000, B 0.000, C 0.000 }
gfCNCPoint3[5537] = {X 143.7791, Y 102.1600, Z -3.8333, A 0.000, B 0.000, C 0.000 }
gfCNCPoint3[5538] = {X 125.0000, Y 102.1600, Z -3.8333, A 0.000, B 0.000, C 0.000 }
gfCNCPoint3[5539] = {X 124.0743, Y 102.0557, Z -3.8333, A 0.000, B 0.000, C 0.000 }
gfCNCPoint3[5540] = {X 123.1950, Y 101.7480, Z -3.8333, A 0.000, B 0.000, C 0.000 }
gfCNCPoint3[5541] = {X 122.4063, Y 101.2524, Z -3.8333, A 0.000, B 0.000, C 0.000 }
gfCNCPoint3[5542] = {X 121.7476, Y 100.5937, Z -3.8333, A 0.000, B 0.000, C 0.000 }
gfCNCPoint3[5543] = {X 121.2520, Y 99.8050, Z -3.8333, A 0.000, B 0.000, C 0.000 }
gfCNCPoint3[5544] = {X 120.9443, Y 98.9257, Z -3.8333, A 0.000, B 0.000, C 0.000 }
gfCNCPoint3[5545] = {X 120.8400, Y 98.0000, Z -3.8333, A 0.000, B 0.000, C 0.000 }
gfCNCPoint3[5546] = {X 120.8400, Y 97.0659, Z -3.8333, A 0.000, B 0.000, C 0.000 }
gfCNCPoint3[5547] = {X 120.9406, Y 96.1566, Z -3.8333, A 0.000, B 0.000, C 0.000 }
gfCNCPoint3[5548] = {X 121.2375, Y 95.2913, Z -3.8333, A 0.000, B 0.000, C 0.000 }
gfCNCPoint3[5549] = {X 121.7164, Y 94.5118, Z -3.8333, A 0.000, B 0.000, C 0.000 }
gfCNCPoint3[5550] = {X 122.3541, Y 93.8558, Z -3.8333, A 0.000, B 0.000, C 0.000 }
gfCNCPoint3[5551] = {X 123.1198, Y 93.3551, Z -3.8333, A 0.000, B 0.000, C 0.000 }
gfCNCPoint3[5552] = {X 123.9764, Y 93.0338, Z -3.8333, A 0.000, B 0.000, C 0.000 }
gfCNCPoint3[5553] = {X 124.8825, Y 92.9076, Z -3.8333, A 0.000, B 0.000, C 0.000 }
gfCNCPoint3[5554] = {X 124.9153, Y 92.8898, Z -3.8333, A 0.000, B 0.000, C 0.000 }
gfCNCPoint3[5555] = {X 124.9514, Y 92.8801, Z -3.8333, A 0.000, B 0.000, C 0.000 }
gfCNCPoint3[5556] = {X 125.4717, Y 92.8029, Z -3.8333, A 0.000, B 0.000, C 0.000 }
gfCNCPoint3[5557] = {X 126.3315, Y 92.6575, Z -3.8333, A 0.000, B 0.000, C 0.000 }
gfCNCPoint3[5558] = {X 127.1790, Y 92.4523, Z -3.8333, A 0.000, B 0.000, C 0.000 }
gfCNCPoint3[5559] = {X 128.4216, Y 91.2831, Z -3.8333, A 0.000, B 0.000, C 0.000 }
gfCNCPoint3[5560] = {X 129.5981, Y 90.0473, Z -3.8333, A 0.000, B 0.000, C 0.000 }
gfCNCPoint3[5561] = {X 140.7986, Y 77.7477, Z -3.8333, A 0.000, B 0.000, C 0.000 }
gfCNCPoint3[5562] = {X 137.8411, Y 75.0545, Z -3.8333, A 0.000, B 0.000, C 0.000 }
gfCNCPoint3[5563] = {X 140.8577, Y 77.8016, Z -3.8333, A 0.000, B 0.000, C 0.000 }
gfCNCPoint3[5564] = {X 155.9352, Y 61.2445, Z -3.8333, A 0.000, B 0.000, C 0.000 }
gfCNCPoint3[5565] = {X 155.5465, Y 60.5382, Z -3.8333, A 0.000, B 0.000, C 0.000 }
gfCNCPoint3[5566] = {X 155.3044, Y 59.7693, Z -3.8333, A 0.000, B 0.000, C 0.000 }
gfCNCPoint3[5567] = {X 155.2181, Y 58.9678, Z -3.8333, A 0.000, B 0.000, C 0.000 }
gfCNCPoint3[5568] = {X 155.2180, Y 58.0000, Z -3.8333, A 0.000, B 0.000, C 0.000 }
gfCNCPoint3[5569] = {X 155.3203, Y 57.0921, Z -3.8333, A 0.000, B 0.000, C 0.000 }
gfCNCPoint3[5570] = {X 155.6220, Y 56.2298, Z -3.8333, A 0.000, B 0.000, C 0.000 }
gfCNCPoint3[5571] = {X 156.1081, Y 55.4562, Z -3.8333, A 0.000, B 0.000, C 0.000 }
gfCNCPoint3[5572] = {X 156.7541, Y 54.8101, Z -3.8333, A 0.000, B 0.000, C 0.000 }
gfCNCPoint3[5573] = {X 157.5277, Y 54.3240, Z -3.8333, A 0.000, B 0.000, C 0.000 }
gfCNCPoint3[5574] = {X 158.3901, Y 54.0223, Z -3.8333, A 0.000, B 0.000, C 0.000 }
gfCNCPoint3[5575] = {X 159.2980, Y 53.9200, Z -3.8333, A 0.000, B 0.000, C 0.000 }
gfCNCPoint3[5576] = {X 178.5335, Y 53.9200, Z -3.8333, A 0.000, B 0.000, C 0.000 }
gfCNCPoint3[5577] = {X 179.4414, Y 54.0223, Z -3.8333, A 0.000, B 0.000, C 0.000 }
gfCNCPoint3[5578] = {X 180.3037, Y 54.3240, Z -3.8333, A 0.000, B 0.000, C 0.000 }
gfCNCPoint3[5579] = {X 181.0773, Y 54.8101, Z -3.8333, A 0.000, B 0.000, C 0.000 }
gfCNCPoint3[5580] = {X 181.7234, Y 55.4562, Z -3.8333, A 0.000, B 0.000, C 0.000 }
gfCNCPoint3[5581] = {X 182.2095, Y 56.2298, Z -3.8333, A 0.000, B 0.000, C 0.000 }
gfCNCPoint3[5582] = {X 182.5112, Y 57.0921, Z -3.8333, A 0.000, B 0.000, C 0.000 }
gfCNCPoint3[5583] = {X 182.6135, Y 58.0000, Z -3.8333, A 0.000, B 0.000, C 0.000 }
gfCNCPoint3[5584] = {X 182.6135, Y 58.9342, Z -3.8333, A 0.000, B 0.000, C 0.000 }
gfCNCPoint3[5585] = {X 182.5334, Y 59.7384, Z -3.8333, A 0.000, B 0.000, C 0.000 }
gfCNCPoint3[5586] = {X 182.2964, Y 60.5111, Z -3.8333, A 0.000, B 0.000, C 0.000 }
gfCNCPoint3[5587] = {X 181.9117, Y 61.2219, Z -3.8333, A 0.000, B 0.000, C 0.000 }
gfCNCPoint3[5588] = {X 209.3014, Y 91.1162, Z -3.8333, A 0.000, B 0.000, C 0.000 }
gfCNCPoint3[5589] = {X 209.9711, Y 91.7957, Z -3.8333, A 0.000, B 0.000, C 0.000 }
gfCNCPoint3[5590] = {X 210.6886, Y 92.4246, Z -3.8333, A 0.000, B 0.000, C 0.000 }
gfCNCPoint3[5591] = {X 211.0136, Y 92.6298, Z -3.8333, A 0.000, B 0.000, C 0.000 }
gfCNCPoint3[5592] = {X 211.3782, Y 92.7518, Z -3.8333, A 0.000, B 0.000, C 0.000 }
gfCNCPoint3[5593] = {X 213.3971, Y 93.0667, Z -3.8333, A 0.000, B 0.000, C 0.000 }
gfCNCPoint3[5594] = {X 214.4548, Y 92.9767, Z -3.8333, A 0.000, B 0.000, C 0.000 }
gfCNCPoint3[5595] = {X 215.5145, Y 92.9158, Z -3.8333, A 0.000, B 0.000, C 0.000 }
gfCNCPoint3[5596] = {X 216.2276, Y 92.8374, Z -3.8333, A 0.000, B 0.000, C 0.000 }
gfCNCPoint3[5597] = {X 216.9142, Y 92.6294, Z -3.8333, A 0.000, B 0.000, C 0.000 }
gfCNCPoint3[5598] = {X 217.5510, Y 92.2991, Z -3.8333, A 0.000, B 0.000, C 0.000 }
gfCNCPoint3[5599] = {X 223.0910, Y 88.7239, Z -3.8333, A 0.000, B 0.000, C 0.000 }
gfCNCPoint3[5600] = {X 246.3544, Y 73.8481, Z -3.8333, A 0.000, B 0.000, C 0.000 }
gfCNCPoint3[5601] = {X 221.7196, Y 64.1805, Z -3.8333, A 0.000, B 0.000, C 0.000 }
gfCNCPoint3[5602] = {X 219.9262, Y 63.5801, Z -3.8333, A 0.000, B 0.000, C 0.000 }
gfCNCPoint3[5603] = {X 218.0759, Y 63.1888, Z -3.8333, A 0.000, B 0.000, C 0.000 }
gfCNCPoint3[5604] = {X 216.1929, Y 63.0117, Z -3.8333, A 0.000, B 0.000, C 0.000 }
gfCNCPoint3[5605] = {X 215.3127, Y 62.8850, Z -3.8333, A 0.000, B 0.000, C 0.000 }
gfCNCPoint3[5606] = {X 214.4809, Y 62.5706, Z -3.8333, A 0.000, B 0.000, C 0.000 }
gfCNCPoint3[5607] = {X 213.7370, Y 62.0834, Z -3.8333, A 0.000, B 0.000, C 0.000 }
gfCNCPoint3[5608] = {X 213.1162, Y 61.4466, Z -3.8333, A 0.000, B 0.000, C 0.000 }
gfCNCPoint3[5609] = {X 212.6482, Y 60.6905, Z -3.8333, A 0.000, B 0.000, C 0.000 }
gfCNCPoint3[5610] = {X 212.3552, Y 59.8509, Z -3.8333, A 0.000, B 0.000, C 0.000 }
gfCNCPoint3[5611] = {X 212.2509, Y 58.9678, Z -3.8333, A 0.000, B 0.000, C 0.000 }
gfCNCPoint3[5612] = {X 212.2508, Y 58.0000, Z -3.8333, A 0.000, B 0.000, C 0.000 }
gfCNCPoint3[5613] = {X 212.3531, Y 57.0921, Z -3.8333, A 0.000, B 0.000, C 0.000 }
gfCNCPoint3[5614] = {X 212.6549, Y 56.2298, Z -3.8333, A 0.000, B 0.000, C 0.000 }
gfCNCPoint3[5615] = {X 213.1409, Y 55.4562, Z -3.8333, A 0.000, B 0.000, C 0.000 }
gfCNCPoint3[5616] = {X 213.7870, Y 54.8101, Z -3.8333, A 0.000, B 0.000, C 0.000 }
gfCNCPoint3[5617] = {X 214.5606, Y 54.3240, Z -3.8333, A 0.000, B 0.000, C 0.000 }
gfCNCPoint3[5618] = {X 215.4229, Y 54.0223, Z -3.8333, A 0.000, B 0.000, C 0.000 }
gfCNCPoint3[5619] = {X 216.3308, Y 53.9200, Z -3.8333, A 0.000, B 0.000, C 0.000 }
gfCNCPoint3[5620] = {X 237.2617, Y 53.9200, Z -3.8333, A 0.000, B 0.000, C 0.000 }
gfCNCPoint3[5621] = {X 238.1696, Y 54.0223, Z -3.8333, A 0.000, B 0.000, C 0.000 }
gfCNCPoint3[5622] = {X 239.0319, Y 54.3240, Z -3.8333, A 0.000, B 0.000, C 0.000 }
gfCNCPoint3[5623] = {X 239.8055, Y 54.8101, Z -3.8333, A 0.000, B 0.000, C 0.000 }
gfCNCPoint3[5624] = {X 240.4516, Y 55.4562, Z -3.8333, A 0.000, B 0.000, C 0.000 }
gfCNCPoint3[5625] = {X 240.9376, Y 56.2298, Z -3.8333, A 0.000, B 0.000, C 0.000 }
gfCNCPoint3[5626] = {X 241.2394, Y 57.0921, Z -3.8333, A 0.000, B 0.000, C 0.000 }
gfCNCPoint3[5627] = {X 241.3417, Y 58.0000, Z -3.8333, A 0.000, B 0.000, C 0.000 }
gfCNCPoint3[5628] = {X 241.3417, Y 58.3965, Z -3.8333, A 0.000, B 0.000, C 0.000 }
gfCNCPoint3[5629] = {X 247.4005, Y 60.7583, Z -3.8333, A 0.000, B 0.000, C 0.000 }
gfCNCPoint3[5630] = {X 275.8731, Y 72.0559, Z -3.8333, A 0.000, B 0.000, C 0.000 }
gfCNCPoint3[5631] = {X 275.8741, Y 62.9983, Z -3.8333, A 0.000, B 0.000, C 0.000 }
gfCNCPoint3[5632] = {X 275.7378, Y 62.9839, Z -3.8333, A 0.000, B 0.000, C 0.000 }
gfCNCPoint3[5633] = {X 275.6020, Y 62.9650, Z -3.8333, A 0.000, B 0.000, C 0.000 }
gfCNCPoint3[5634] = {X 274.6824, Y 62.7081, Z -3.8333, A 0.000, B 0.000, C 0.000 }
gfCNCPoint3[5635] = {X 273.8478, Y 62.2444, Z -3.8333, A 0.000, B 0.000, C 0.000 }
gfCNCPoint3[5636] = {X 273.1437, Y 61.5995, Z -3.8333, A 0.000, B 0.000, C 0.000 }
gfCNCPoint3[5637] = {X 272.6088, Y 60.8086, Z -3.8333, A 0.000, B 0.000, C 0.000 }
gfCNCPoint3[5638] = {X 272.2724, Y 59.9150, Z -3.8333, A 0.000, B 0.000, C 0.000 }
gfCNCPoint3[5639] = {X 272.1528, Y 58.9678, Z -3.8333, A 0.000, B 0.000, C 0.000 }
gfCNCPoint3[5640] = {X 272.1527, Y 58.0000, Z -3.8333, A 0.000, B 0.000, C 0.000 }
gfCNCPoint3[5641] = {X 272.2550, Y 57.0921, Z -3.8333, A 0.000, B 0.000, C 0.000 }
gfCNCPoint3[5642] = {X 272.5567, Y 56.2298, Z -3.8333, A 0.000, B 0.000, C 0.000 }
gfCNCPoint3[5643] = {X 273.0428, Y 55.4562, Z -3.8333, A 0.000, B 0.000, C 0.000 }
gfCNCPoint3[5644] = {X 273.6889, Y 54.8101, Z -3.8333, A 0.000, B 0.000, C 0.000 }
gfCNCPoint3[5645] = {X 274.4624, Y 54.3240, Z -3.8333, A 0.000, B 0.000, C 0.000 }
gfCNCPoint3[5646] = {X 275.3248, Y 54.0223, Z -3.8333, A 0.000, B 0.000, C 0.000 }
gfCNCPoint3[5647] = {X 276.2327, Y 53.9200, Z -3.8333, A 0.000, B 0.000, C 0.000 }
gfCNCPoint3[5648] = {X 292.7731, Y 53.9200, Z -3.8333, A 0.000, B 0.000, C 0.000 }
gfCNCPoint3[5649] = {X 293.6810, Y 54.0223, Z -3.8333, A 0.000, B 0.000, C 0.000 }
gfCNCPoint3[5650] = {X 294.5433, Y 54.3240, Z -3.8333, A 0.000, B 0.000, C 0.000 }
gfCNCPoint3[5651] = {X 295.3169, Y 54.8101, Z -3.8333, A 0.000, B 0.000, C 0.000 }
gfCNCPoint3[5652] = {X 295.9630, Y 55.4562, Z -3.8333, A 0.000, B 0.000, C 0.000 }
gfCNCPoint3[5653] = {X 296.4490, Y 56.2298, Z -3.8333, A 0.000, B 0.000, C 0.000 }
gfCNCPoint3[5654] = {X 296.7508, Y 57.0921, Z -3.8333, A 0.000, B 0.000, C 0.000 }
gfCNCPoint3[5655] = {X 296.8531, Y 58.0000, Z -3.8333, A 0.000, B 0.000, C 0.000 }
gfCNCPoint3[5656] = {X 296.8531, Y 58.9344, Z -3.8333, A 0.000, B 0.000, C 0.000 }
gfCNCPoint3[5657] = {X 296.7375, Y 59.8874, Z -3.8333, A 0.000, B 0.000, C 0.000 }
gfCNCPoint3[5658] = {X 296.4033, Y 60.7874, Z -3.8333, A 0.000, B 0.000, C 0.000 }
gfCNCPoint3[5659] = {X 295.8688, Y 61.5849, Z -3.8333, A 0.000, B 0.000, C 0.000 }
gfCNCPoint3[5660] = {X 295.1634, Y 62.2361, Z -3.8333, A 0.000, B 0.000, C 0.000 }
gfCNCPoint3[5661] = {X 294.3258, Y 62.7053, Z -3.8333, A 0.000, B 0.000, C 0.000 }
gfCNCPoint3[5662] = {X 293.4020, Y 62.9666, Z -3.8333, A 0.000, B 0.000, C 0.000 }
gfCNCPoint3[5663] = {X 293.2754, Y 62.9848, Z -3.8333, A 0.000, B 0.000, C 0.000 }
gfCNCPoint3[5664] = {X 293.1482, Y 62.9990, Z -3.8333, A 0.000, B 0.000, C 0.000 }
gfCNCPoint3[5665] = {X 293.1324, Y 63.1580, Z -3.8333, A 0.000, B 0.000, C 0.000 }
gfCNCPoint3[5666] = {X 293.1445, Y 92.9934, Z -3.8333, A 0.000, B 0.000, C 0.000 }
gfCNCPoint3[5667] = {X 293.2730, Y 93.0082, Z -3.8333, A 0.000, B 0.000, C 0.000 }
gfCNCPoint3[5668] = {X 293.4010, Y 93.0269, Z -3.8333, A 0.000, B 0.000, C 0.000 }
gfCNCPoint3[5669] = {X 294.3245, Y 93.2909, Z -3.8333, A 0.000, B 0.000, C 0.000 }
gfCNCPoint3[5670] = {X 295.1617, Y 93.7618, Z -3.8333, A 0.000, B 0.000, C 0.000 }
gfCNCPoint3[5671] = {X 295.8667, Y 94.4141, Z -3.8333, A 0.000, B 0.000, C 0.000 }
gfCNCPoint3[5672] = {X 296.4013, Y 95.2121, Z -3.8333, A 0.000, B 0.000, C 0.000 }
gfCNCPoint3[5673] = {X 296.7361, Y 96.1123, Z -3.8333, A 0.000, B 0.000, C 0.000 }
gfCNCPoint3[5674] = {X 296.8531, Y 97.0657, Z -3.8333, A 0.000, B 0.000, C 0.000 }
gfCNCPoint3[5675] = {X 296.8531, Y 98.0000, Z -3.8333, A 0.000, B 0.000, C 0.000 }
gfCNCPoint3[5676] = {X 296.7508, Y 98.9079, Z -3.8333, A 0.000, B 0.000, C 0.000 }
gfCNCPoint3[5677] = {X 296.4490, Y 99.7702, Z -3.8333, A 0.000, B 0.000, C 0.000 }
gfCNCPoint3[5678] = {X 295.9630, Y 100.5438, Z -3.8333, A 0.000, B 0.000, C 0.000 }
gfCNCPoint3[5679] = {X 295.3169, Y 101.1899, Z -3.8333, A 0.000, B 0.000, C 0.000 }
gfCNCPoint3[5680] = {X 294.5433, Y 101.6760, Z -3.8333, A 0.000, B 0.000, C 0.000 }
gfCNCPoint3[5681] = {X 293.6810, Y 101.9777, Z -3.8333, A 0.000, B 0.000, C 0.000 }
gfCNCPoint3[5682] = {X 292.7731, Y 102.0800, Z -3.8333, A 0.000, B 0.000, C 0.000 }
gfCNCPoint3[5683] = {X 276.2327, Y 102.0800, Z -3.8333, A 0.000, B 0.000, C 0.000 }
gfCNCPoint3[5684] = {X 275.3248, Y 101.9777, Z -3.8333, A 0.000, B 0.000, C 0.000 }
gfCNCPoint3[5685] = {X 274.4624, Y 101.6760, Z -3.8333, A 0.000, B 0.000, C 0.000 }
gfCNCPoint3[5686] = {X 273.6889, Y 101.1899, Z -3.8333, A 0.000, B 0.000, C 0.000 }
gfCNCPoint3[5687] = {X 273.0428, Y 100.5438, Z -3.8333, A 0.000, B 0.000, C 0.000 }
gfCNCPoint3[5688] = {X 272.5567, Y 99.7702, Z -3.8333, A 0.000, B 0.000, C 0.000 }
gfCNCPoint3[5689] = {X 272.2550, Y 98.9079, Z -3.8333, A 0.000, B 0.000, C 0.000 }
gfCNCPoint3[5690] = {X 272.1527, Y 98.0000, Z -3.8333, A 0.000, B 0.000, C 0.000 }
gfCNCPoint3[5691] = {X 272.1527, Y 97.0659, Z -3.8333, A 0.000, B 0.000, C 0.000 }
gfCNCPoint3[5692] = {X 272.2437, Y 96.2088, Z -3.8333, A 0.000, B 0.000, C 0.000 }
gfCNCPoint3[5693] = {X 272.5128, Y 95.3899, Z -3.8333, A 0.000, B 0.000, C 0.000 }
gfCNCPoint3[5694] = {X 272.9480, Y 94.6458, Z -3.8333, A 0.000, B 0.000, C 0.000 }
gfCNCPoint3[5695] = {X 273.5297, Y 94.0097, Z -3.8333, A 0.000, B 0.000, C 0.000 }
gfCNCPoint3[5696] = {X 274.2321, Y 93.5101, Z -3.8333, A 0.000, B 0.000, C 0.000 }
gfCNCPoint3[5697] = {X 275.0238, Y 93.1692, Z -3.8333, A 0.000, B 0.000, C 0.000 }
gfCNCPoint3[5698] = {X 275.8694, Y 93.0021, Z -3.8333, A 0.000, B 0.000, C 0.000 }
gfCNCPoint3[5699] = {X 275.8694, Y 85.4313, Z -3.8333, A 0.000, B 0.000, C 0.000 }
gfCNCPoint3[5700] = {X 262.6143, Y 80.2353, Z -3.8333, A 0.000, B 0.000, C 0.000 }
gfCNCPoint3[5701] = {X 262.1474, Y 80.5294, Z -3.8333, A 0.000, B 0.000, C 0.000 }
gfCNCPoint3[5702] = {X 237.5555, Y 96.4582, Z -3.8333, A 0.000, B 0.000, C 0.000 }
gfCNCPoint3[5703] = {X 237.5598, Y 97.0656, Z -3.8333, A 0.000, B 0.000, C 0.000 }
gfCNCPoint3[5704] = {X 237.5598, Y 98.0000, Z -3.8333, A 0.000, B 0.000, C 0.000 }
gfCNCPoint3[5705] = {X 237.4575, Y 98.9079, Z -3.8333, A 0.000, B 0.000, C 0.000 }
gfCNCPoint3[5706] = {X 237.1557, Y 99.7702, Z -3.8333, A 0.000, B 0.000, C 0.000 }
gfCNCPoint3[5707] = {X 236.6697, Y 100.5438, Z -3.8333, A 0.000, B 0.000, C 0.000 }
gfCNCPoint3[5708] = {X 236.0236, Y 101.1899, Z -3.8333, A 0.000, B 0.000, C 0.000 }
gfCNCPoint3[5709] = {X 235.2500, Y 101.6760, Z -3.8333, A 0.000, B 0.000, C 0.000 }
gfCNCPoint3[5710] = {X 234.3877, Y 101.9777, Z -3.8333, A 0.000, B 0.000, C 0.000 }
gfCNCPoint3[5711] = {X 233.4798, Y 102.0800, Z -3.8333, A 0.000, B 0.000, C 0.000 }
gfCNCPoint3[5712] = {X 214.1790, Y 102.0800, Z -3.8333, A 0.000, B 0.000, C 0.000 }
gfCNCPoint3[5713] = {X 213.7860, Y 102.0610, Z -3.8333, A 0.000, B 0.000, C 0.000 }
gfCNCPoint3[5714] = {X 213.3966, Y 102.0043, Z -3.8333, A 0.000, B 0.000, C 0.000 }
gfCNCPoint3[5715] = {X 213.0072, Y 102.0610, Z -3.8333, A 0.000, B 0.000, C 0.000 }
gfCNCPoint3[5716] = {X 212.6141, Y 102.0800, Z -3.8333, A 0.000, B 0.000, C 0.000 }
gfCNCPoint3[5717] = {X 194.9870, Y 102.0800, Z -3.8333, A 0.000, B 0.000, C 0.000 }
gfCNCPoint3[5718] = {X 194.0791, Y 101.9777, Z -3.8333, A 0.000, B 0.000, C 0.000 }
gfCNCPoint3[5719] = {X 193.2167, Y 101.6760, Z -3.8333, A 0.000, B 0.000, C 0.000 }
gfCNCPoint3[5720] = {X 192.4431, Y 101.1899, Z -3.8333, A 0.000, B 0.000, C 0.000 }
gfCNCPoint3[5721] = {X 191.7971, Y 100.5438, Z -3.8333, A 0.000, B 0.000, C 0.000 }
gfCNCPoint3[5722] = {X 191.3110, Y 99.7702, Z -3.8333, A 0.000, B 0.000, C 0.000 }
gfCNCPoint3[5723] = {X 191.0093, Y 98.9079, Z -3.8333, A 0.000, B 0.000, C 0.000 }
gfCNCPoint3[5724] = {X 190.9070, Y 98.0000, Z -3.8333, A 0.000, B 0.000, C 0.000 }
gfCNCPoint3[5725] = {X 190.9070, Y 97.0659, Z -3.8333, A 0.000, B 0.000, C 0.000 }
gfCNCPoint3[5726] = {X 191.0022, Y 96.1894, Z -3.8333, A 0.000, B 0.000, C 0.000 }
gfCNCPoint3[5727] = {X 191.2835, Y 95.3539, Z -3.8333, A 0.000, B 0.000, C 0.000 }
gfCNCPoint3[5728] = {X 191.7378, Y 94.5983, Z -3.8333, A 0.000, B 0.000, C 0.000 }
gfCNCPoint3[5729] = {X 191.8199, Y 94.4938, Z -3.8333, A 0.000, B 0.000, C 0.000 }
gfCNCPoint3[5730] = {X 191.9053, Y 94.3920, Z -3.8333, A 0.000, B 0.000, C 0.000 }
gfCNCPoint3[5731] = {X 188.6703, Y 90.8602, Z -3.8333, A 0.000, B 0.000, C 0.000 }
gfCNCPoint3[5732] = {X 149.9831, Y 90.8602, Z -3.8333, A 0.000, B 0.000, C 0.000 }
gfCNCPoint3[5733] = {X 146.8265, Y 94.3574, Z -3.8333, A 0.000, B 0.000, C 0.000 }
gfCNCPoint3[5734] = {X 147.3864, Y 95.1679, Z -3.8333, A 0.000, B 0.000, C 0.000 }
gfCNCPoint3[5735] = {X 147.7374, Y 96.0883, Z -3.8333, A 0.000, B 0.000, C 0.000 }
gfCNCPoint3[5736] = {X 147.8591, Y 97.0658, Z -3.8333, A 0.000, B 0.000, C 0.000 }
gfCNCPoint3[5737] = {X 147.8591, Y 98.0000, Z -3.8333, A 0.000, B 0.000, C 0.000 }
gfCNCPoint3[5738] = {X 147.7568, Y 98.9079, Z -3.8333, A 0.000, B 0.000, C 0.000 }
gfCNCPoint3[5739] = {X 147.4551, Y 99.7702, Z -3.8333, A 0.000, B 0.000, C 0.000 }
gfCNCPoint3[5740] = {X 146.9690, Y 100.5438, Z -3.8333, A 0.000, B 0.000, C 0.000 }
gfCNCPoint3[5741] = {X 146.3229, Y 101.1899, Z -3.8333, A 0.000, B 0.000, C 0.000 }
gfCNCPoint3[5742] = {X 145.5494, Y 101.6760, Z -3.8333, A 0.000, B 0.000, C 0.000 }
gfCNCPoint3[5743] = {X 144.6870, Y 101.9777, Z -3.8333, A 0.000, B 0.000, C 0.000 }
gfCNCPoint3[5744] = {X 143.7791, Y 102.0800, Z -3.8333, A 0.000, B 0.000, C 0.000 }
gfCNCPoint3[5745] = {X 125.0000, Y 102.0800, Z -3.8333, A 0.000, B 0.000, C 0.000 }
gfCNCPoint3[5746] = {X 124.0921, Y 101.9777, Z -3.8333, A 0.000, B 0.000, C 0.000 }
gfCNCPoint3[5747] = {X 123.2298, Y 101.6760, Z -3.8333, A 0.000, B 0.000, C 0.000 }
gfCNCPoint3[5748] = {X 122.4562, Y 101.1899, Z -3.8333, A 0.000, B 0.000, C 0.000 }
gfCNCPoint3[5749] = {X 121.8101, Y 100.5438, Z -3.8333, A 0.000, B 0.000, C 0.000 }
gfCNCPoint3[5750] = {X 121.3240, Y 99.7702, Z -3.8333, A 0.000, B 0.000, C 0.000 }
gfCNCPoint3[5751] = {X 121.0223, Y 98.9079, Z -3.8333, A 0.000, B 0.000, C 0.000 }
gfCNCPoint3[5752] = {X 120.9200, Y 98.0000, Z -3.8333, A 0.000, B 0.000, C 0.000 }
gfCNCPoint3[5753] = {X 120.9200, Y 97.0659, Z -3.8333, A 0.000, B 0.000, C 0.000 }
gfCNCPoint3[5754] = {X 121.0194, Y 96.1710, Z -3.8333, A 0.000, B 0.000, C 0.000 }
gfCNCPoint3[5755] = {X 121.3126, Y 95.3196, Z -3.8333, A 0.000, B 0.000, C 0.000 }
gfCNCPoint3[5756] = {X 121.7855, Y 94.5532, Z -3.8333, A 0.000, B 0.000, C 0.000 }
gfCNCPoint3[5757] = {X 122.4150, Y 93.9093, Z -3.8333, A 0.000, B 0.000, C 0.000 }
gfCNCPoint3[5758] = {X 123.1704, Y 93.4192, Z -3.8333, A 0.000, B 0.000, C 0.000 }
gfCNCPoint3[5759] = {X 124.0149, Y 93.1066, Z -3.8333, A 0.000, B 0.000, C 0.000 }
gfCNCPoint3[5760] = {X 124.9074, Y 92.9870, Z -3.8333, A 0.000, B 0.000, C 0.000 }
gfCNCPoint3[5761] = {X 124.9308, Y 92.9715, Z -3.8333, A 0.000, B 0.000, C 0.000 }
gfCNCPoint3[5762] = {X 124.9631, Y 92.9592, Z -3.8333, A 0.000, B 0.000, C 0.000 }
gfCNCPoint3[5763] = {X 125.4829, Y 92.8821, Z -3.8333, A 0.000, B 0.000, C 0.000 }
gfCNCPoint3[5764] = {X 126.3570, Y 92.7339, Z -3.8333, A 0.000, B 0.000, C 0.000 }
gfCNCPoint3[5765] = {X 127.2184, Y 92.5244, Z -3.8333, A 0.000, B 0.000, C 0.000 }
gfCNCPoint3[5766] = {X 128.4714, Y 91.3463, Z -3.8333, A 0.000, B 0.000, C 0.000 }
gfCNCPoint3[5767] = {X 129.6575, Y 90.1009, Z -3.8333, A 0.000, B 0.000, C 0.000 }
gfCNCPoint3[5768] = {X 140.8577, Y 77.8016, Z -3.8333, A 0.000, B 0.000, C 0.000 }
gfCNCPoint3[5769] = {X 137.8976, Y 75.1061, Z -3.8333, A 0.000, B 0.000, C 0.000 }
gfCNCPoint3[5770] = {X 137.8980, Y 75.1056, Z -3.8333, A 0.000, B 0.000, C 0.000 }
gfCNCPoint3[5771] = {X 140.9143, Y 77.8531, Z -3.8333, A 0.000, B 0.000, C 0.000 }
gfCNCPoint3[5772] = {X 156.0374, Y 61.2511, Z -3.8333, A 0.000, B 0.000, C 0.000 }
gfCNCPoint3[5773] = {X 155.6325, Y 60.5354, Z -3.8333, A 0.000, B 0.000, C 0.000 }
gfCNCPoint3[5774] = {X 155.3825, Y 59.7520, Z -3.8333, A 0.000, B 0.000, C 0.000 }
gfCNCPoint3[5775] = {X 155.2980, Y 58.9340, Z -3.8333, A 0.000, B 0.000, C 0.000 }
gfCNCPoint3[5776] = {X 155.2980, Y 58.0000, Z -3.8333, A 0.000, B 0.000, C 0.000 }
gfCNCPoint3[5777] = {X 155.3982, Y 57.1099, Z -3.8333, A 0.000, B 0.000, C 0.000 }
gfCNCPoint3[5778] = {X 155.6941, Y 56.2645, Z -3.8333, A 0.000, B 0.000, C 0.000 }
gfCNCPoint3[5779] = {X 156.1706, Y 55.5060, Z -3.8333, A 0.000, B 0.000, C 0.000 }
gfCNCPoint3[5780] = {X 156.8040, Y 54.8727, Z -3.8333, A 0.000, B 0.000, C 0.000 }
gfCNCPoint3[5781] = {X 157.5624, Y 54.3961, Z -3.8333, A 0.000, B 0.000, C 0.000 }
gfCNCPoint3[5782] = {X 158.4079, Y 54.1003, Z -3.8333, A 0.000, B 0.000, C 0.000 }
gfCNCPoint3[5783] = {X 159.2980, Y 54.0000, Z -3.8333, A 0.000, B 0.000, C 0.000 }
gfCNCPoint3[5784] = {X 178.5335, Y 54.0000, Z -3.8333, A 0.000, B 0.000, C 0.000 }
gfCNCPoint3[5785] = {X 179.4236, Y 54.1003, Z -3.8333, A 0.000, B 0.000, C 0.000 }
gfCNCPoint3[5786] = {X 180.2690, Y 54.3961, Z -3.8333, A 0.000, B 0.000, C 0.000 }
gfCNCPoint3[5787] = {X 181.0275, Y 54.8727, Z -3.8333, A 0.000, B 0.000, C 0.000 }
gfCNCPoint3[5788] = {X 181.6608, Y 55.5060, Z -3.8333, A 0.000, B 0.000, C 0.000 }
gfCNCPoint3[5789] = {X 182.1374, Y 56.2645, Z -3.8333, A 0.000, B 0.000, C 0.000 }
gfCNCPoint3[5790] = {X 182.4332, Y 57.1099, Z -3.8333, A 0.000, B 0.000, C 0.000 }
gfCNCPoint3[5791] = {X 182.5335, Y 58.0000, Z -3.8333, A 0.000, B 0.000, C 0.000 }
gfCNCPoint3[5792] = {X 182.5334, Y 58.9671, Z -3.8333, A 0.000, B 0.000, C 0.000 }
gfCNCPoint3[5793] = {X 182.4463, Y 59.7647, Z -3.8333, A 0.000, B 0.000, C 0.000 }
gfCNCPoint3[5794] = {X 182.2018, Y 60.5289, Z -3.8333, A 0.000, B 0.000, C 0.000 }
gfCNCPoint3[5795] = {X 181.8097, Y 61.2290, Z -3.8333, A 0.000, B 0.000, C 0.000 }
gfCNCPoint3[5796] = {X 209.2424, Y 91.1702, Z -3.8333, A 0.000, B 0.000, C 0.000 }
gfCNCPoint3[5797] = {X 209.9162, Y 91.8539, Z -3.8333, A 0.000, B 0.000, C 0.000 }
gfCNCPoint3[5798] = {X 210.6381, Y 92.4867, Z -3.8333, A 0.000, B 0.000, C 0.000 }
gfCNCPoint3[5799] = {X 210.9793, Y 92.7021, Z -3.8333, A 0.000, B 0.000, C 0.000 }
gfCNCPoint3[5800] = {X 211.3621, Y 92.8301, Z -3.8333, A 0.000, B 0.000, C 0.000 }
gfCNCPoint3[5801] = {X 212.0545, Y 92.9782, Z -3.8333, A 0.000, B 0.000, C 0.000 }
gfCNCPoint3[5802] = {X 213.3960, Y 93.1472, Z -3.8333, A 0.000, B 0.000, C 0.000 }
gfCNCPoint3[5803] = {X 214.4554, Y 93.0569, Z -3.8333, A 0.000, B 0.000, C 0.000 }
gfCNCPoint3[5804] = {X 215.5170, Y 92.9958, Z -3.8333, A 0.000, B 0.000, C 0.000 }
gfCNCPoint3[5805] = {X 216.2444, Y 92.9156, Z -3.8333, A 0.000, B 0.000, C 0.000 }
gfCNCPoint3[5806] = {X 216.9448, Y 92.7034, Z -3.8333, A 0.000, B 0.000, C 0.000 }
gfCNCPoint3[5807] = {X 217.5944, Y 92.3663, Z -3.8333, A 0.000, B 0.000, C 0.000 }
gfCNCPoint3[5808] = {X 223.1343, Y 88.7912, Z -3.8333, A 0.000, B 0.000, C 0.000 }
gfCNCPoint3[5809] = {X 246.5297, Y 73.8310, Z -3.8333, A 0.000, B 0.000, C 0.000 }
gfCNCPoint3[5810] = {X 221.7493, Y 64.1062, Z -3.8333, A 0.000, B 0.000, C 0.000 }
gfCNCPoint3[5811] = {X 219.9472, Y 63.5029, Z -3.8333, A 0.000, B 0.000, C 0.000 }
gfCNCPoint3[5812] = {X 218.0879, Y 63.1097, Z -3.8333, A 0.000, B 0.000, C 0.000 }
gfCNCPoint3[5813] = {X 216.1958, Y 62.9318, Z -3.8333, A 0.000, B 0.000, C 0.000 }
gfCNCPoint3[5814] = {X 215.3283, Y 62.8064, Z -3.8333, A 0.000, B 0.000, C 0.000 }
gfCNCPoint3[5815] = {X 214.5089, Y 62.4950, Z -3.8333, A 0.000, B 0.000, C 0.000 }
gfCNCPoint3[5816] = {X 213.7770, Y 62.0127, Z -3.8333, A 0.000, B 0.000, C 0.000 }
gfCNCPoint3[5817] = {X 213.1677, Y 61.3825, Z -3.8333, A 0.000, B 0.000, C 0.000 }
gfCNCPoint3[5818] = {X 212.7104, Y 60.6348, Z -3.8333, A 0.000, B 0.000, C 0.000 }
gfCNCPoint3[5819] = {X 212.4268, Y 59.8053, Z -3.8333, A 0.000, B 0.000, C 0.000 }
gfCNCPoint3[5820] = {X 212.3308, Y 58.9340, Z -3.8333, A 0.000, B 0.000, C 0.000 }
gfCNCPoint3[5821] = {X 212.3308, Y 58.0000, Z -3.8333, A 0.000, B 0.000, C 0.000 }
gfCNCPoint3[5822] = {X 212.4311, Y 57.1099, Z -3.8333, A 0.000, B 0.000, C 0.000 }
gfCNCPoint3[5823] = {X 212.7269, Y 56.2645, Z -3.8333, A 0.000, B 0.000, C 0.000 }
gfCNCPoint3[5824] = {X 213.2035, Y 55.5060, Z -3.8333, A 0.000, B 0.000, C 0.000 }
gfCNCPoint3[5825] = {X 213.8368, Y 54.8727, Z -3.8333, A 0.000, B 0.000, C 0.000 }
gfCNCPoint3[5826] = {X 214.5953, Y 54.3961, Z -3.8333, A 0.000, B 0.000, C 0.000 }
gfCNCPoint3[5827] = {X 215.4407, Y 54.1003, Z -3.8333, A 0.000, B 0.000, C 0.000 }
gfCNCPoint3[5828] = {X 216.3308, Y 54.0000, Z -3.8333, A 0.000, B 0.000, C 0.000 }
gfCNCPoint3[5829] = {X 237.2617, Y 54.0000, Z -3.8333, A 0.000, B 0.000, C 0.000 }
gfCNCPoint3[5830] = {X 238.1518, Y 54.1003, Z -3.8333, A 0.000, B 0.000, C 0.000 }
gfCNCPoint3[5831] = {X 238.9972, Y 54.3961, Z -3.8333, A 0.000, B 0.000, C 0.000 }
gfCNCPoint3[5832] = {X 239.7556, Y 54.8727, Z -3.8333, A 0.000, B 0.000, C 0.000 }
gfCNCPoint3[5833] = {X 240.3890, Y 55.5060, Z -3.8333, A 0.000, B 0.000, C 0.000 }
gfCNCPoint3[5834] = {X 240.8656, Y 56.2645, Z -3.8333, A 0.000, B 0.000, C 0.000 }
gfCNCPoint3[5835] = {X 241.1614, Y 57.1099, Z -3.8333, A 0.000, B 0.000, C 0.000 }
gfCNCPoint3[5836] = {X 241.2617, Y 58.0000, Z -3.8333, A 0.000, B 0.000, C 0.000 }
gfCNCPoint3[5837] = {X 241.2617, Y 58.4512, Z -3.8333, A 0.000, B 0.000, C 0.000 }
gfCNCPoint3[5838] = {X 247.3712, Y 60.8328, Z -3.8333, A 0.000, B 0.000, C 0.000 }
gfCNCPoint3[5839] = {X 275.9532, Y 72.1737, Z -3.8333, A 0.000, B 0.000, C 0.000 }
gfCNCPoint3[5840] = {X 275.9525, Y 63.0385, Z -3.8333, A 0.000, B 0.000, C 0.000 }
gfCNCPoint3[5841] = {X 275.9573, Y 62.9246, Z -3.8333, A 0.000, B 0.000, C 0.000 }
gfCNCPoint3[5842] = {X 275.7854, Y 62.9090, Z -3.8333, A 0.000, B 0.000, C 0.000 }
gfCNCPoint3[5843] = {X 275.6144, Y 62.8860, Z -3.8333, A 0.000, B 0.000, C 0.000 }
gfCNCPoint3[5844] = {X 274.7077, Y 62.6320, Z -3.8333, A 0.000, B 0.000, C 0.000 }
gfCNCPoint3[5845] = {X 273.8856, Y 62.1731, Z -3.8333, A 0.000, B 0.000, C 0.000 }
gfCNCPoint3[5846] = {X 273.1935, Y 61.5347, Z -3.8333, A 0.000, B 0.000, C 0.000 }
gfCNCPoint3[5847] = {X 272.6698, Y 60.7522, Z -3.8333, A 0.000, B 0.000, C 0.000 }
gfCNCPoint3[5848] = {X 272.3435, Y 59.8691, Z -3.8333, A 0.000, B 0.000, C 0.000 }
gfCNCPoint3[5849] = {X 272.2327, Y 58.9340, Z -3.8333, A 0.000, B 0.000, C 0.000 }
gfCNCPoint3[5850] = {X 272.2327, Y 58.0000, Z -3.8333, A 0.000, B 0.000, C 0.000 }
gfCNCPoint3[5851] = {X 272.3330, Y 57.1099, Z -3.8333, A 0.000, B 0.000, C 0.000 }
gfCNCPoint3[5852] = {X 272.6288, Y 56.2645, Z -3.8333, A 0.000, B 0.000, C 0.000 }
gfCNCPoint3[5853] = {X 273.1054, Y 55.5060, Z -3.8333, A 0.000, B 0.000, C 0.000 }
gfCNCPoint3[5854] = {X 273.7387, Y 54.8727, Z -3.8333, A 0.000, B 0.000, C 0.000 }
gfCNCPoint3[5855] = {X 274.4972, Y 54.3961, Z -3.8333, A 0.000, B 0.000, C 0.000 }
gfCNCPoint3[5856] = {X 275.3426, Y 54.1003, Z -3.8333, A 0.000, B 0.000, C 0.000 }
gfCNCPoint3[5857] = {X 276.2327, Y 54.0000, Z -3.8333, A 0.000, B 0.000, C 0.000 }
gfCNCPoint3[5858] = {X 292.7731, Y 54.0000, Z -3.8333, A 0.000, B 0.000, C 0.000 }
gfCNCPoint3[5859] = {X 293.6632, Y 54.1003, Z -3.8333, A 0.000, B 0.000, C 0.000 }
gfCNCPoint3[5860] = {X 294.5086, Y 54.3961, Z -3.8333, A 0.000, B 0.000, C 0.000 }
gfCNCPoint3[5861] = {X 295.2670, Y 54.8727, Z -3.8333, A 0.000, B 0.000, C 0.000 }
gfCNCPoint3[5862] = {X 295.9004, Y 55.5060, Z -3.8333, A 0.000, B 0.000, C 0.000 }
gfCNCPoint3[5863] = {X 296.3770, Y 56.2645, Z -3.8333, A 0.000, B 0.000, C 0.000 }
gfCNCPoint3[5864] = {X 296.6728, Y 57.1099, Z -3.8333, A 0.000, B 0.000, C 0.000 }
gfCNCPoint3[5865] = {X 296.7731, Y 58.0000, Z -3.8333, A 0.000, B 0.000, C 0.000 }
gfCNCPoint3[5866] = {X 296.7731, Y 58.9341, Z -3.8333, A 0.000, B 0.000, C 0.000 }
gfCNCPoint3[5867] = {X 296.6598, Y 59.8685, Z -3.8333, A 0.000, B 0.000, C 0.000 }
gfCNCPoint3[5868] = {X 296.3321, Y 60.7510, Z -3.8333, A 0.000, B 0.000, C 0.000 }
gfCNCPoint3[5869] = {X 295.8080, Y 61.5329, Z -3.8333, A 0.000, B 0.000, C 0.000 }
gfCNCPoint3[5870] = {X 295.1164, Y 62.1714, Z -3.8333, A 0.000, B 0.000, C 0.000 }
gfCNCPoint3[5871] = {X 294.2952, Y 62.6314, Z -3.8333, A 0.000, B 0.000, C 0.000 }
gfCNCPoint3[5872] = {X 293.3894, Y 62.8876, Z -3.8333, A 0.000, B 0.000, C 0.000 }
gfCNCPoint3[5873] = {X 293.2327, Y 62.9094, Z -3.8333, A 0.000, B 0.000, C 0.000 }
gfCNCPoint3[5874] = {X 293.0752, Y 62.9251, Z -3.8333, A 0.000, B 0.000, C 0.000 }
gfCNCPoint3[5875] = {X 293.0524, Y 63.1540, Z -3.8333, A 0.000, B 0.000, C 0.000 }
gfCNCPoint3[5876] = {X 293.0524, Y 92.9237, Z -3.8333, A 0.000, B 0.000, C 0.000 }
gfCNCPoint3[5877] = {X 293.0752, Y 93.0675, Z -3.8333, A 0.000, B 0.000, C 0.000 }
gfCNCPoint3[5878] = {X 293.2320, Y 93.0836, Z -3.8333, A 0.000, B 0.000, C 0.000 }
gfCNCPoint3[5879] = {X 293.3882, Y 93.1059, Z -3.8333, A 0.000, B 0.000, C 0.000 }
gfCNCPoint3[5880] = {X 294.2937, Y 93.3647, Z -3.8333, A 0.000, B 0.000, C 0.000 }
gfCNCPoint3[5881] = {X 295.1146, Y 93.8265, Z -3.8333, A 0.000, B 0.000, C 0.000 }
gfCNCPoint3[5882] = {X 295.8059, Y 94.4661, Z -3.8333, A 0.000, B 0.000, C 0.000 }
gfCNCPoint3[5883] = {X 296.3300, Y 95.2486, Z -3.8333, A 0.000, B 0.000, C 0.000 }
gfCNCPoint3[5884] = {X 296.6584, Y 96.1313, Z -3.8333, A 0.000, B 0.000, C 0.000 }
gfCNCPoint3[5885] = {X 296.7731, Y 97.0661, Z -3.8333, A 0.000, B 0.000, C 0.000 }
gfCNCPoint3[5886] = {X 296.7731, Y 98.0000, Z -3.8333, A 0.000, B 0.000, C 0.000 }
gfCNCPoint3[5887] = {X 296.6728, Y 98.8901, Z -3.8333, A 0.000, B 0.000, C 0.000 }
gfCNCPoint3[5888] = {X 296.3770, Y 99.7355, Z -3.8333, A 0.000, B 0.000, C 0.000 }
gfCNCPoint3[5889] = {X 295.9004, Y 100.4940, Z -3.8333, A 0.000, B 0.000, C 0.000 }
gfCNCPoint3[5890] = {X 295.2670, Y 101.1273, Z -3.8333, A 0.000, B 0.000, C 0.000 }
gfCNCPoint3[5891] = {X 294.5086, Y 101.6039, Z -3.8333, A 0.000, B 0.000, C 0.000 }
gfCNCPoint3[5892] = {X 293.6632, Y 101.8997, Z -3.8333, A 0.000, B 0.000, C 0.000 }
gfCNCPoint3[5893] = {X 292.7731, Y 102.0000, Z -3.8333, A 0.000, B 0.000, C 0.000 }
gfCNCPoint3[5894] = {X 276.2327, Y 102.0000, Z -3.8333, A 0.000, B 0.000, C 0.000 }
gfCNCPoint3[5895] = {X 275.3426, Y 101.8997, Z -3.8333, A 0.000, B 0.000, C 0.000 }
gfCNCPoint3[5896] = {X 274.4972, Y 101.6039, Z -3.8333, A 0.000, B 0.000, C 0.000 }
gfCNCPoint3[5897] = {X 273.7387, Y 101.1273, Z -3.8333, A 0.000, B 0.000, C 0.000 }
gfCNCPoint3[5898] = {X 273.1054, Y 100.4940, Z -3.8333, A 0.000, B 0.000, C 0.000 }
gfCNCPoint3[5899] = {X 272.6288, Y 99.7355, Z -3.8333, A 0.000, B 0.000, C 0.000 }
gfCNCPoint3[5900] = {X 272.3330, Y 98.8901, Z -3.8333, A 0.000, B 0.000, C 0.000 }
gfCNCPoint3[5901] = {X 272.2327, Y 98.0000, Z -3.8333, A 0.000, B 0.000, C 0.000 }
gfCNCPoint3[5902] = {X 272.2329, Y 97.0232, Z -3.8333, A 0.000, B 0.000, C 0.000 }
gfCNCPoint3[5903] = {X 272.3321, Y 96.1797, Z -3.8333, A 0.000, B 0.000, C 0.000 }
gfCNCPoint3[5904] = {X 272.6072, Y 95.3761, Z -3.8333, A 0.000, B 0.000, C 0.000 }
gfCNCPoint3[5905] = {X 273.0457, Y 94.6486, Z -3.8333, A 0.000, B 0.000, C 0.000 }
gfCNCPoint3[5906] = {X 273.6280, Y 94.0302, Z -3.8333, A 0.000, B 0.000, C 0.000 }
gfCNCPoint3[5907] = {X 274.3277, Y 93.5487, Z -3.8333, A 0.000, B 0.000, C 0.000 }
gfCNCPoint3[5908] = {X 275.1133, Y 93.2258, Z -3.8333, A 0.000, B 0.000, C 0.000 }
gfCNCPoint3[5909] = {X 275.9494, Y 93.0760, Z -3.8333, A 0.000, B 0.000, C 0.000 }
gfCNCPoint3[5910] = {X 275.9494, Y 85.3767, Z -3.8333, A 0.000, B 0.000, C 0.000 }
gfCNCPoint3[5911] = {X 262.6059, Y 80.1460, Z -3.8333, A 0.000, B 0.000, C 0.000 }
gfCNCPoint3[5912] = {X 262.1044, Y 80.4620, Z -3.8333, A 0.000, B 0.000, C 0.000 }
gfCNCPoint3[5913] = {X 237.4752, Y 96.4149, Z -3.8333, A 0.000, B 0.000, C 0.000 }
gfCNCPoint3[5914] = {X 237.4798, Y 97.0659, Z -3.8333, A 0.000, B 0.000, C 0.000 }
gfCNCPoint3[5915] = {X 237.4798, Y 98.0000, Z -3.8333, A 0.000, B 0.000, C 0.000 }
gfCNCPoint3[5916] = {X 237.3795, Y 98.8901, Z -3.8333, A 0.000, B 0.000, C 0.000 }
gfCNCPoint3[5917] = {X 237.0837, Y 99.7355, Z -3.8333, A 0.000, B 0.000, C 0.000 }
gfCNCPoint3[5918] = {X 236.6071, Y 100.4940, Z -3.8333, A 0.000, B 0.000, C 0.000 }
gfCNCPoint3[5919] = {X 235.9737, Y 101.1273, Z -3.8333, A 0.000, B 0.000, C 0.000 }
gfCNCPoint3[5920] = {X 235.2153, Y 101.6039, Z -3.8333, A 0.000, B 0.000, C 0.000 }
gfCNCPoint3[5921] = {X 234.3699, Y 101.8997, Z -3.8333, A 0.000, B 0.000, C 0.000 }
gfCNCPoint3[5922] = {X 233.4798, Y 102.0000, Z -3.8333, A 0.000, B 0.000, C 0.000 }
gfCNCPoint3[5923] = {X 214.1790, Y 102.0000, Z -3.8333, A 0.000, B 0.000, C 0.000 }
gfCNCPoint3[5924] = {X 213.7859, Y 101.9806, Z -3.8333, A 0.000, B 0.000, C 0.000 }
gfCNCPoint3[5925] = {X 213.3966, Y 101.9227, Z -3.8333, A 0.000, B 0.000, C 0.000 }
gfCNCPoint3[5926] = {X 213.0072, Y 101.9806, Z -3.8333, A 0.000, B 0.000, C 0.000 }
gfCNCPoint3[5927] = {X 212.6141, Y 102.0000, Z -3.8333, A 0.000, B 0.000, C 0.000 }
gfCNCPoint3[5928] = {X 194.9870, Y 102.0000, Z -3.8333, A 0.000, B 0.000, C 0.000 }
gfCNCPoint3[5929] = {X 194.0969, Y 101.8997, Z -3.8333, A 0.000, B 0.000, C 0.000 }
gfCNCPoint3[5930] = {X 193.2514, Y 101.6039, Z -3.8333, A 0.000, B 0.000, C 0.000 }
gfCNCPoint3[5931] = {X 192.4930, Y 101.1273, Z -3.8333, A 0.000, B 0.000, C 0.000 }
gfCNCPoint3[5932] = {X 191.8596, Y 100.4940, Z -3.8333, A 0.000, B 0.000, C 0.000 }
gfCNCPoint3[5933] = {X 191.3831, Y 99.7355, Z -3.8333, A 0.000, B 0.000, C 0.000 }
gfCNCPoint3[5934] = {X 191.0872, Y 98.8901, Z -3.8333, A 0.000, B 0.000, C 0.000 }
gfCNCPoint3[5935] = {X 190.9870, Y 98.0000, Z -3.8333, A 0.000, B 0.000, C 0.000 }
gfCNCPoint3[5936] = {X 190.9870, Y 97.0659, Z -3.8333, A 0.000, B 0.000, C 0.000 }
gfCNCPoint3[5937] = {X 191.0804, Y 96.2066, Z -3.8333, A 0.000, B 0.000, C 0.000 }
gfCNCPoint3[5938] = {X 191.3562, Y 95.3874, Z -3.8333, A 0.000, B 0.000, C 0.000 }
gfCNCPoint3[5939] = {X 191.8015, Y 94.6466, Z -3.8333, A 0.000, B 0.000, C 0.000 }
gfCNCPoint3[5940] = {X 191.9056, Y 94.5177, Z -3.8333, A 0.000, B 0.000, C 0.000 }
gfCNCPoint3[5941] = {X 192.0149, Y 94.3932, Z -3.8333, A 0.000, B 0.000, C 0.000 }
gfCNCPoint3[5942] = {X 188.7055, Y 90.7802, Z -3.8333, A 0.000, B 0.000, C 0.000 }
gfCNCPoint3[5943] = {X 149.9476, Y 90.7802, Z -3.8333, A 0.000, B 0.000, C 0.000 }
gfCNCPoint3[5944] = {X 146.7187, Y 94.3574, Z -3.8333, A 0.000, B 0.000, C 0.000 }
gfCNCPoint3[5945] = {X 147.1685, Y 94.9488, Z -3.8333, A 0.000, B 0.000, C 0.000 }
gfCNCPoint3[5946] = {X 147.5020, Y 95.6127, Z -3.8333, A 0.000, B 0.000, C 0.000 }
gfCNCPoint3[5947] = {X 147.7079, Y 96.3266, Z -3.8333, A 0.000, B 0.000, C 0.000 }
gfCNCPoint3[5948] = {X 147.7791, Y 97.0661, Z -3.8333, A 0.000, B 0.000, C 0.000 }
gfCNCPoint3[5949] = {X 147.7791, Y 98.0000, Z -3.8333, A 0.000, B 0.000, C 0.000 }
gfCNCPoint3[5950] = {X 147.6788, Y 98.8901, Z -3.8333, A 0.000, B 0.000, C 0.000 }
gfCNCPoint3[5951] = {X 147.3830, Y 99.7355, Z -3.8333, A 0.000, B 0.000, C 0.000 }
gfCNCPoint3[5952] = {X 146.9064, Y 100.4940, Z -3.8333, A 0.000, B 0.000, C 0.000 }
gfCNCPoint3[5953] = {X 146.2731, Y 101.1273, Z -3.8333, A 0.000, B 0.000, C 0.000 }
gfCNCPoint3[5954] = {X 145.5146, Y 101.6039, Z -3.8333, A 0.000, B 0.000, C 0.000 }
gfCNCPoint3[5955] = {X 144.6692, Y 101.8997, Z -3.8333, A 0.000, B 0.000, C 0.000 }
gfCNCPoint3[5956] = {X 143.7791, Y 102.0000, Z -3.8333, A 0.000, B 0.000, C 0.000 }
gfCNCPoint3[5957] = {X 125.0000, Y 102.0000, Z -3.8333, A 0.000, B 0.000, C 0.000 }
gfCNCPoint3[5958] = {X 124.1099, Y 101.8997, Z -3.8333, A 0.000, B 0.000, C 0.000 }
gfCNCPoint3[5959] = {X 123.2645, Y 101.6039, Z -3.8333, A 0.000, B 0.000, C 0.000 }
gfCNCPoint3[5960] = {X 122.5060, Y 101.1273, Z -3.8333, A 0.000, B 0.000, C 0.000 }
gfCNCPoint3[5961] = {X 121.8727, Y 100.4940, Z -3.8333, A 0.000, B 0.000, C 0.000 }
gfCNCPoint3[5962] = {X 121.3961, Y 99.7355, Z -3.8333, A 0.000, B 0.000, C 0.000 }
gfCNCPoint3[5963] = {X 121.1003, Y 98.8901, Z -3.8333, A 0.000, B 0.000, C 0.000 }
gfCNCPoint3[5964] = {X 121.0000, Y 98.0000, Z -3.8333, A 0.000, B 0.000, C 0.000 }
gfCNCPoint3[5965] = {X 121.0000, Y 97.0659, Z -3.8333, A 0.000, B 0.000, C 0.000 }
gfCNCPoint3[5966] = {X 121.0981, Y 96.1853, Z -3.8333, A 0.000, B 0.000, C 0.000 }
gfCNCPoint3[5967] = {X 121.3877, Y 95.3479, Z -3.8333, A 0.000, B 0.000, C 0.000 }
gfCNCPoint3[5968] = {X 121.8546, Y 94.5948, Z -3.8333, A 0.000, B 0.000, C 0.000 }
gfCNCPoint3[5969] = {X 122.4758, Y 93.9629, Z -3.8333, A 0.000, B 0.000, C 0.000 }
gfCNCPoint3[5970] = {X 123.2209, Y 93.4834, Z -3.8333, A 0.000, B 0.000, C 0.000 }
gfCNCPoint3[5971] = {X 124.0533, Y 93.1796, Z -3.8333, A 0.000, B 0.000, C 0.000 }
gfCNCPoint3[5972] = {X 124.9321, Y 93.0665, Z -3.8333, A 0.000, B 0.000, C 0.000 }
gfCNCPoint3[5973] = {X 124.9749, Y 93.0383, Z -3.8333, A 0.000, B 0.000, C 0.000 }
gfCNCPoint3[5974] = {X 125.4940, Y 92.9613, Z -3.8333, A 0.000, B 0.000, C 0.000 }
gfCNCPoint3[5975] = {X 126.3824, Y 92.8104, Z -3.8333, A 0.000, B 0.000, C 0.000 }
gfCNCPoint3[5976] = {X 127.2578, Y 92.5964, Z -3.8333, A 0.000, B 0.000, C 0.000 }
gfCNCPoint3[5977] = {X 128.5213, Y 91.4095, Z -3.8333, A 0.000, B 0.000, C 0.000 }
gfCNCPoint3[5978] = {X 129.7170, Y 90.1544, Z -3.8333, A 0.000, B 0.000, C 0.000 }
gfCNCPoint3[5979] = {X 133.8038, Y 85.6588, Z -3.8333, A 0.000, B 0.000, C 0.000 }
gfCNCPoint3[5980] = {X 140.9143, Y 77.8531, Z -3.8333, A 0.000, B 0.000, C 0.000 }
gfCNCPoint3[5981] = {X 137.8980, Y 75.1056, Z -3.8333, A 0.000, B 0.000, C 0.000 }
gfCNCPoint3[5982] = {X 137.8980, Y 75.1056, Z -0.8333, A 0.000, B 0.000, C 0.000 }
gfCNCPoint3[5983] = {X 137.8980, Y 75.1056, Z 11.0000, A 0.000, B 0.000, C 0.000 }
gfCNCPoint3[5984] = {X 167.3809, Y 20.2812, Z 11.0000, A 0.000, B 0.000, C 0.000 }
gfCNCPoint3[5985] = {X 167.3809, Y 20.2812, Z -0.8333, A 0.000, B 0.000, C 0.000 }
gfCNCPoint3[5986] = {X 167.3809, Y 20.2812, Z -3.8333, A 0.000, B 0.000, C 0.000 }
gfCNCPoint3[5987] = {X 171.1581, Y 18.7388, Z -3.8333, A 0.000, B 0.000, C 0.000 }
gfCNCPoint3[5988] = {X 169.8405, Y 15.5121, Z -3.8333, A 0.000, B 0.000, C 0.000 }
gfCNCPoint3[5989] = {X 169.5912, Y 14.6607, Z -3.8333, A 0.000, B 0.000, C 0.000 }
gfCNCPoint3[5990] = {X 169.5212, Y 13.7764, Z -3.8333, A 0.000, B 0.000, C 0.000 }
gfCNCPoint3[5991] = {X 169.6332, Y 12.8964, Z -3.8333, A 0.000, B 0.000, C 0.000 }
gfCNCPoint3[5992] = {X 169.9226, Y 12.0578, Z -3.8333, A 0.000, B 0.000, C 0.000 }
gfCNCPoint3[5993] = {X 170.3773, Y 11.2960, Z -3.8333, A 0.000, B 0.000, C 0.000 }
gfCNCPoint3[5994] = {X 170.9779, Y 10.6432, Z -3.8333, A 0.000, B 0.000, C 0.000 }
gfCNCPoint3[5995] = {X 171.6992, Y 10.1268, Z -3.8333, A 0.000, B 0.000, C 0.000 }
gfCNCPoint3[5996] = {X 172.3295, Y 9.7674, Z -3.8333, A 0.000, B 0.000, C 0.000 }
gfCNCPoint3[5997] = {X 173.2114, Y 9.3960, Z -3.8333, A 0.000, B 0.000, C 0.000 }
gfCNCPoint3[5998] = {X 174.1534, Y 9.2278, Z -3.8333, A 0.000, B 0.000, C 0.000 }
gfCNCPoint3[5999] = {X 175.1093, Y 9.2711, Z -3.8333, A 0.000, B 0.000, C 0.000 }
gfCNCPoint3[6000] = {X 176.0322, Y 9.5238, Z -3.8333, A 0.000, B 0.000, C 0.000 }
gfCNCPoint3[6001] = {X 178.2250, Y 8.6010, Z -3.8333, A 0.000, B 0.000, C 0.000 }
gfCNCPoint3[6002] = {X 180.4990, Y 7.9023, Z -3.8333, A 0.000, B 0.000, C 0.000 }
gfCNCPoint3[6003] = {X 182.8315, Y 7.4345, Z -3.8333, A 0.000, B 0.000, C 0.000 }
gfCNCPoint3[6004] = {X 185.1991, Y 7.2025, Z -3.8333, A 0.000, B 0.000, C 0.000 }
gfCNCPoint3[6005] = {X 187.5781, Y 7.2084, Z -3.8333, A 0.000, B 0.000, C 0.000 }
gfCNCPoint3[6006] = {X 189.9445, Y 7.4523, Z -3.8333, A 0.000, B 0.000, C 0.000 }
gfCNCPoint3[6007] = {X 191.7018, Y 7.8137, Z -3.8333, A 0.000, B 0.000, C 0.000 }
gfCNCPoint3[6008] = {X 193.4127, Y 8.3536, Z -3.8333, A 0.000, B 0.000, C 0.000 }
gfCNCPoint3[6009] = {X 195.0591, Y 9.0664, Z -3.8333, A 0.000, B 0.000, C 0.000 }
gfCNCPoint3[6010] = {X 196.6236, Y 9.9444, Z -3.8333, A 0.000, B 0.000, C 0.000 }
gfCNCPoint3[6011] = {X 198.0897, Y 10.9785, Z -3.8333, A 0.000, B 0.000, C 0.000 }
gfCNCPoint3[6012] = {X 199.1492, Y 11.9219, Z -3.8333, A 0.000, B 0.000, C 0.000 }
gfCNCPoint3[6013] = {X 200.1001, Y 12.9747, Z -3.8333, A 0.000, B 0.000, C 0.000 }
gfCNCPoint3[6014] = {X 200.9311, Y 14.1246, Z -3.8333, A 0.000, B 0.000, C 0.000 }
gfCNCPoint3[6015] = {X 201.6324, Y 15.3578, Z -3.8333, A 0.000, B 0.000, C 0.000 }
gfCNCPoint3[6016] = {X 202.1957, Y 16.6598, Z -3.8333, A 0.000, B 0.000, C 0.000 }
gfCNCPoint3[6017] = {X 202.6699, Y 18.3162, Z -3.8333, A 0.000, B 0.000, C 0.000 }
gfCNCPoint3[6018] = {X 202.9514, Y 20.0159, Z -3.8333, A 0.000, B 0.000, C 0.000 }
gfCNCPoint3[6019] = {X 203.0364, Y 21.7367, Z -3.8333, A 0.000, B 0.000, C 0.000 }
gfCNCPoint3[6020] = {X 202.9238, Y 23.4559, Z -3.8333, A 0.000, B 0.000, C 0.000 }
gfCNCPoint3[6021] = {X 202.6151, Y 25.1510, Z -3.8333, A 0.000, B 0.000, C 0.000 }
gfCNCPoint3[6022] = {X 202.1733, Y 26.5971, Z -3.8333, A 0.000, B 0.000, C 0.000 }
gfCNCPoint3[6023] = {X 201.5486, Y 27.9741, Z -3.8333, A 0.000, B 0.000, C 0.000 }
gfCNCPoint3[6024] = {X 200.7514, Y 29.2590, Z -3.8333, A 0.000, B 0.000, C 0.000 }
gfCNCPoint3[6025] = {X 199.7950, Y 30.4303, Z -3.8333, A 0.000, B 0.000, C 0.000 }
gfCNCPoint3[6026] = {X 198.6955, Y 31.4683, Z -3.8333, A 0.000, B 0.000, C 0.000 }
gfCNCPoint3[6027] = {X 199.4969, Y 31.8095, Z -3.8333, A 0.000, B 0.000, C 0.000 }
gfCNCPoint3[6028] = {X 200.2135, Y 32.3045, Z -3.8333, A 0.000, B 0.000, C 0.000 }
gfCNCPoint3[6029] = {X 200.8164, Y 32.9333, Z -3.8333, A 0.000, B 0.000, C 0.000 }
gfCNCPoint3[6030] = {X 201.2808, Y 33.6702, Z -3.8333, A 0.000, B 0.000, C 0.000 }
gfCNCPoint3[6031] = {X 204.3222, Y 39.9530, Z -3.8333, A 0.000, B 0.000, C 0.000 }
gfCNCPoint3[6032] = {X 204.6427, Y 40.8622, Z -3.8333, A 0.000, B 0.000, C 0.000 }
gfCNCPoint3[6033] = {X 204.7537, Y 41.8197, Z -3.8333, A 0.000, B 0.000, C 0.000 }
gfCNCPoint3[6034] = {X 204.6496, Y 42.7781, Z -3.8333, A 0.000, B 0.000, C 0.000 }
gfCNCPoint3[6035] = {X 204.3355, Y 43.6895, Z -3.8333, A 0.000, B 0.000, C 0.000 }
gfCNCPoint3[6036] = {X 203.8272, Y 44.5085, Z -3.8333, A 0.000, B 0.000, C 0.000 }
gfCNCPoint3[6037] = {X 203.1499, Y 45.1945, Z -3.8333, A 0.000, B 0.000, C 0.000 }
gfCNCPoint3[6038] = {X 202.6136, Y 45.6281, Z -3.8333, A 0.000, B 0.000, C 0.000 }
gfCNCPoint3[6039] = {X 201.9090, Y 46.0917, Z -3.8333, A 0.000, B 0.000, C 0.000 }
gfCNCPoint3[6040] = {X 201.1279, Y 46.4100, Z -3.8333, A 0.000, B 0.000, C 0.000 }
gfCNCPoint3[6041] = {X 200.2999, Y 46.5710, Z -3.8333, A 0.000, B 0.000, C 0.000 }
gfCNCPoint3[6042] = {X 199.4564, Y 46.5686, Z -3.8333, A 0.000, B 0.000, C 0.000 }
gfCNCPoint3[6043] = {X 198.6294, Y 46.4028, Z -3.8333, A 0.000, B 0.000, C 0.000 }
gfCNCPoint3[6044] = {X 196.2990, Y 47.6051, Z -3.8333, A 0.000, B 0.000, C 0.000 }
gfCNCPoint3[6045] = {X 193.8686, Y 48.5897, Z -3.8333, A 0.000, B 0.000, C 0.000 }
gfCNCPoint3[6046] = {X 191.3585, Y 49.3484, Z -3.8333, A 0.000, B 0.000, C 0.000 }
gfCNCPoint3[6047] = {X 189.4154, Y 49.7421, Z -3.8333, A 0.000, B 0.000, C 0.000 }
gfCNCPoint3[6048] = {X 187.4454, Y 49.9644, Z -3.8333, A 0.000, B 0.000, C 0.000 }
gfCNCPoint3[6049] = {X 185.4634, Y 50.0136, Z -3.8333, A 0.000, B 0.000, C 0.000 }
gfCNCPoint3[6050] = {X 183.4847, Y 49.8893, Z -3.8333, A 0.000, B 0.000, C 0.000 }
gfCNCPoint3[6051] = {X 181.5245, Y 49.5924, Z -3.8333, A 0.000, B 0.000, C 0.000 }
gfCNCPoint3[6052] = {X 179.6380, Y 49.1208, Z -3.8333, A 0.000, B 0.000, C 0.000 }
gfCNCPoint3[6053] = {X 177.8176, Y 48.4373, Z -3.8333, A 0.000, B 0.000, C 0.000 }
gfCNCPoint3[6054] = {X 176.0869, Y 47.5509, Z -3.8333, A 0.000, B 0.000, C 0.000 }
gfCNCPoint3[6055] = {X 174.4685, Y 46.4729, Z -3.8333, A 0.000, B 0.000, C 0.000 }
gfCNCPoint3[6056] = {X 173.2357, Y 45.4324, Z -3.8333, A 0.000, B 0.000, C 0.000 }
gfCNCPoint3[6057] = {X 172.1387, Y 44.2496, Z -3.8333, A 0.000, B 0.000, C 0.000 }
gfCNCPoint3[6058] = {X 171.1937, Y 42.9422, Z -3.8333, A 0.000, B 0.000, C 0.000 }
gfCNCPoint3[6059] = {X 170.4148, Y 41.5295, Z -3.8333, A 0.000, B 0.000, C 0.000 }
gfCNCPoint3[6060] = {X 169.8135, Y 40.0325, Z -3.8333, A 0.000, B 0.000, C 0.000 }
gfCNCPoint3[6061] = {X 169.3988, Y 38.4735, Z -3.8333, A 0.000, B 0.000, C 0.000 }
gfCNCPoint3[6062] = {X 169.1769, Y 36.8756, Z -3.8333, A 0.000, B 0.000, C 0.000 }
gfCNCPoint3[6063] = {X 169.0929, Y 35.0416, Z -3.8333, A 0.000, B 0.000, C 0.000 }
